LIN {X 0,Y 581.296,Z 726.906,A -85,B 0,C 180,E1 9487.47,E2 9487.47} C_VEL
LIN {X 0,Y 571.469,Z 707.643,A -85,B 0,C 180,E1 9488.58,E2 9488.58} C_VEL
LIN {X 0,Y 571.367,Z 707.31,A -85,B 0,C 180,E1 9494.263,E2 9494.263} C_VEL
LIN {X 0,Y 571.407,Z 707.31,A -85,B 0,C 180,E1 9500.466,E2 9500.466} C_VEL
LIN {X 0,Y 571.477,Z 707.31,A -85,B 0,C 180,E1 9506.158,E2 9506.158} C_VEL
LIN {X 0,Y 571.546,Z 707.31,A -85,B 0,C 180,E1 9511.491,E2 9511.491} C_VEL
LIN {X 0,Y 571.588,Z 707.31,A -85,B 0,C 180,E1 9516.564,E2 9516.564} C_VEL
LIN {X 0,Y 571.677,Z 707.31,A -85,B 0,C 180,E1 9522.611,E2 9522.611} C_VEL
LIN {X 0,Y 572.124,Z 707.31,A -85,B 0,C 180,E1 9528.533,E2 9528.533} C_VEL
LIN {X 0,Y 572.269,Z 707.31,A -85,B 0,C 180,E1 9533.917,E2 9533.917} C_VEL
LIN {X 0,Y 572.201,Z 707.31,A -85,B 0,C 180,E1 9539.997,E2 9539.997} C_VEL
LIN {X 0,Y 572.109,Z 707.31,A -85,B 0,C 180,E1 9546.079,E2 9546.079} C_VEL
LIN {X 0,Y 572.048,Z 707.31,A -85,B 0,C 180,E1 9551.43,E2 9551.43} C_VEL
LIN {X 0,Y 571.675,Z 707.31,A -85,B 0,C 180,E1 9557.388,E2 9557.388} C_VEL
LIN {X 0,Y 571.56,Z 707.31,A -85,B 0,C 180,E1 9563.431,E2 9563.431} C_VEL
LIN {X 0,Y 571.547,Z 707.31,A -85,B 0,C 180,E1 9568.958,E2 9568.958} C_VEL
LIN {X 0,Y 571.47,Z 707.31,A -85,B 0,C 180,E1 9574.709,E2 9574.709} C_VEL
LIN {X 0,Y 571.379,Z 707.31,A -85,B 0,C 180,E1 9579.723,E2 9579.723} C_VEL
LIN {X 0,Y 571.332,Z 707.31,A -85,B 0,C 180,E1 9585.733,E2 9585.733} C_VEL
LIN {X 0,Y 571.387,Z 707.31,A -85,B 0,C 180,E1 9588.976,E2 9588.976} C_VEL
LIN {X 0,Y 578.42,Z 721.819,A -85,B 0,C 180,E1 9589.801,E2 9589.801} C_VEL
LIN {X 0,Y 603.039,Z 770.669,A -85,B 0,C 180,E1 9592.453,E2 9592.453} C_VEL
LIN {X 0,Y 600.05,Z 820.289,A -85,B 0,C 180,E1 9593.653,E2 9593.653} C_VEL
LIN {X 0,Y 598.7,Z 837.933,A -85,B 0,C 180,E1 9594.27,E2 9594.27} C_VEL
LIN {X 0,Y 593.828,Z 854.218,A -85,B 0,C 180,E1 9594.704,E2 9594.704} C_VEL
LIN {X 0,Y 588.685,Z 870.067,A -85,B 0,C 180,E1 9595.207,E2 9595.207} C_VEL
LIN {X 0,Y 583.535,Z 912.903,A -85,B 0,C 180,E1 9597.679,E2 9597.679} C_VEL
LIN {X 0,Y 578.202,Z 952.807,A -85,B 0,C 180,E1 9600.781,E2 9600.781} C_VEL
LIN {X 0,Y 573.288,Z 989.217,A -85,B 0,C 180,E1 9604.529,E2 9604.529} C_VEL
LIN {X 0,Y 569.458,Z 1019.706,A -85,B 0,C 180,E1 9608.644,E2 9608.644} C_VEL
LIN {X 0,Y 566.797,Z 1045.546,A -85,B 0,C 180,E1 9613.296,E2 9613.296} C_VEL
LIN {X 0,Y 565.422,Z 1063.972,A -85,B 0,C 180,E1 9617.923,E2 9617.923} C_VEL
LIN {X 0,Y 564.867,Z 1075.583,A -85,B 0,C 180,E1 9622.291,E2 9622.291} C_VEL
LIN {X 0,Y 564.721,Z 1080.643,A -85,B 0,C 180,E1 9625.382,E2 9625.382} C_VEL
LIN {X 0,Y 564.787,Z 1083.5,A -85,B 0,C 180,E1 9629.999,E2 9629.999} C_VEL
LIN {X 0,Y 564.751,Z 1080.646,A -85,B 0,C 180,E1 9634.617,E2 9634.617} C_VEL
LIN {X 0,Y 564.884,Z 1073.99,A -85,B 0,C 180,E1 9638.484,E2 9638.484} C_VEL
LIN {X 0,Y 565.598,Z 1060.203,A -85,B 0,C 180,E1 9643.163,E2 9643.163} C_VEL
LIN {X 0,Y 567.063,Z 1041.597,A -85,B 0,C 180,E1 9647.495,E2 9647.495} C_VEL
LIN {X 0,Y 569.661,Z 1017.405,A -85,B 0,C 180,E1 9651.696,E2 9651.696} C_VEL
LIN {X 0,Y 573.518,Z 986.806,A -85,B 0,C 180,E1 9655.747,E2 9655.747} C_VEL
LIN {X 0,Y 578.55,Z 950.559,A -85,B 0,C 180,E1 9659.413,E2 9659.413} C_VEL
LIN {X 0,Y 584.004,Z 910.777,A -85,B 0,C 180,E1 9662.474,E2 9662.474} C_VEL
LIN {X 0,Y 589.211,Z 868.238,A -85,B 0,C 180,E1 9664.906,E2 9664.906} C_VEL
LIN {X 0,Y 593.615,Z 824.295,A -85,B 0,C 180,E1 9666.688,E2 9666.688} C_VEL
LIN {X 0,Y 596.654,Z 780.659,A -85,B 0,C 180,E1 9667.85,E2 9667.85} C_VEL
LIN {X 0,Y 596.255,Z 771.433,A -85,B 0,C 180,E1 9668.098,E2 9668.098} C_VEL
LIN {X 0,Y 574.83,Z 728.644,A -85,B 0,C 180,E1 9670.579,E2 9670.579} C_VEL
LIN {X 0,Y 563.718,Z 709.225,A -85,B 0,C 180,E1 9671.902,E2 9671.902} C_VEL
LIN {X 0,Y 563.489,Z 707.31,A -85,B 0,C 180,E1 9672.019,E2 9672.019} C_VEL
LIN {X 0,Y 563.451,Z 707.31,A -85,B 0,C 180,E1 9677.754,E2 9677.754} C_VEL
LIN {X 0,Y 563.526,Z 707.31,A -85,B 0,C 180,E1 9683.778,E2 9683.778} C_VEL
LIN {X 0,Y 563.666,Z 707.31,A -85,B 0,C 180,E1 9689.35,E2 9689.35} C_VEL
LIN {X 0,Y 563.629,Z 707.31,A -85,B 0,C 180,E1 9694.524,E2 9694.524} C_VEL
LIN {X 0,Y 563.692,Z 707.31,A -85,B 0,C 180,E1 9700.205,E2 9700.205} C_VEL
LIN {X 0,Y 563.965,Z 707.31,A -85,B 0,C 180,E1 9706.008,E2 9706.008} C_VEL
LIN {X 0,Y 564.245,Z 707.31,A -85,B 0,C 180,E1 9710.73,E2 9710.73} C_VEL
LIN {X 0,Y 563.991,Z 707.31,A -85,B 0,C 180,E1 9715.379,E2 9715.379} C_VEL
LIN {X 0,Y 564.275,Z 707.31,A -85,B 0,C 180,E1 9720.003,E2 9720.003} C_VEL
LIN {X 0,Y 564.043,Z 707.31,A -85,B 0,C 180,E1 9726.25,E2 9726.25} C_VEL
LIN {X 0,Y 564.054,Z 707.31,A -85,B 0,C 180,E1 9732.414,E2 9732.414} C_VEL
LIN {X 0,Y 563.768,Z 707.31,A -85,B 0,C 180,E1 9738.82,E2 9738.82} C_VEL
LIN {X 0,Y 563.719,Z 707.31,A -85,B 0,C 180,E1 9743.939,E2 9743.939} C_VEL
LIN {X 0,Y 563.492,Z 707.31,A -85,B 0,C 180,E1 9748.955,E2 9748.955} C_VEL
LIN {X 0,Y 563.465,Z 707.31,A -85,B 0,C 180,E1 9754.39,E2 9754.39} C_VEL
LIN {X 0,Y 563.457,Z 707.31,A -85,B 0,C 180,E1 9760.204,E2 9760.204} C_VEL
LIN {X 0,Y 563.487,Z 707.4,A -85,B 0,C 180,E1 9766.379,E2 9766.379} C_VEL
LIN {X 0,Y 568.232,Z 717.353,A -85,B 0,C 180,E1 9766.983,E2 9766.983} C_VEL
LIN {X 0,Y 588.613,Z 755.907,A -85,B 0,C 180,E1 9769.479,E2 9769.479} C_VEL
LIN {X 0,Y 595.824,Z 774.73,A -85,B 0,C 180,E1 9770.57,E2 9770.57} C_VEL
LIN {X 0,Y 591.999,Z 820.472,A -85,B 0,C 180,E1 9772.096,E2 9772.096} C_VEL
LIN {X 0,Y 587.146,Z 862.961,A -85,B 0,C 180,E1 9774.17,E2 9774.17} C_VEL
LIN {X 0,Y 582.133,Z 901.788,A -85,B 0,C 180,E1 9776.757,E2 9776.757} C_VEL
LIN {X 0,Y 576.775,Z 939.323,A -85,B 0,C 180,E1 9780.054,E2 9780.054} C_VEL
LIN {X 0,Y 572.225,Z 972.486,A -85,B 0,C 180,E1 9783.881,E2 9783.881} C_VEL
LIN {X 0,Y 568.66,Z 1000.305,A -85,B 0,C 180,E1 9788.095,E2 9788.095} C_VEL
LIN {X 0,Y 566.274,Z 1023.607,A -85,B 0,C 180,E1 9792.881,E2 9792.881} C_VEL
LIN {X 0,Y 565.16,Z 1039.587,A -85,B 0,C 180,E1 9797.614,E2 9797.614} C_VEL
LIN {X 0,Y 564.745,Z 1049.246,A -85,B 0,C 180,E1 9802.29,E2 9802.29} C_VEL
LIN {X 0,Y 564.561,Z 1053.277,A -85,B 0,C 180,E1 9806.923,E2 9806.923} C_VEL
LIN {X 0,Y 564.853,Z 1052.901,A -85,B 0,C 180,E1 9810.001,E2 9810.001} C_VEL
LIN {X 0,Y 564.793,Z 1047.709,A -85,B 0,C 180,E1 9814.618,E2 9814.618} C_VEL
LIN {X 0,Y 565.152,Z 1037.925,A -85,B 0,C 180,E1 9818.87,E2 9818.87} C_VEL
LIN {X 0,Y 566.241,Z 1023.115,A -85,B 0,C 180,E1 9823.149,E2 9823.149} C_VEL
LIN {X 0,Y 568.566,Z 1000.113,A -85,B 0,C 180,E1 9827.85,E2 9827.85} C_VEL
LIN {X 0,Y 572.256,Z 971.194,A -85,B 0,C 180,E1 9832.202,E2 9832.202} C_VEL
LIN {X 0,Y 577.134,Z 936.917,A -85,B 0,C 180,E1 9836.093,E2 9836.093} C_VEL
LIN {X 0,Y 582.635,Z 897.836,A -85,B 0,C 180,E1 9839.435,E2 9839.435} C_VEL
LIN {X 0,Y 588.021,Z 856.086,A -85,B 0,C 180,E1 9842.09,E2 9842.09} C_VEL
LIN {X 0,Y 592.591,Z 812.427,A -85,B 0,C 180,E1 9844.087,E2 9844.087} C_VEL
LIN {X 0,Y 594.966,Z 772.076,A -85,B 0,C 180,E1 9845.404,E2 9845.404} C_VEL
LIN {X 0,Y 574.604,Z 728.871,A -85,B 0,C 180,E1 9847.981,E2 9847.981} C_VEL
LIN {X 0,Y 563.598,Z 708.617,A -85,B 0,C 180,E1 9849.24,E2 9849.24} C_VEL
LIN {X 0,Y 563.51,Z 707.31,A -85,B 0,C 180,E1 9849.325,E2 9849.325} C_VEL
LIN {X 0,Y 563.489,Z 707.31,A -85,B 0,C 180,E1 9855.632,E2 9855.632} C_VEL
LIN {X 0,Y 563.458,Z 707.31,A -85,B 0,C 180,E1 9861.785,E2 9861.785} C_VEL
LIN {X 0,Y 563.6,Z 707.31,A -85,B 0,C 180,E1 9867.466,E2 9867.466} C_VEL
LIN {X 0,Y 563.638,Z 707.31,A -85,B 0,C 180,E1 9872.8,E2 9872.8} C_VEL
LIN {X 0,Y 563.701,Z 707.31,A -85,B 0,C 180,E1 9877.889,E2 9877.889} C_VEL
LIN {X 0,Y 563.962,Z 707.31,A -85,B 0,C 180,E1 9884.41,E2 9884.41} C_VEL
LIN {X 0,Y 564.262,Z 707.31,A -85,B 0,C 180,E1 9889.162,E2 9889.162} C_VEL
LIN {X 0,Y 564.354,Z 707.31,A -85,B 0,C 180,E1 9895.377,E2 9895.377} C_VEL
LIN {X 0,Y 564.428,Z 707.31,A -85,B 0,C 180,E1 9901.536,E2 9901.536} C_VEL
LIN {X 0,Y 564.373,Z 707.31,A -85,B 0,C 180,E1 9907.713,E2 9907.713} C_VEL
LIN {X 0,Y 564.094,Z 707.31,A -85,B 0,C 180,E1 9912.407,E2 9912.407} C_VEL
LIN {X 0,Y 563.812,Z 707.31,A -85,B 0,C 180,E1 9917.194,E2 9917.194} C_VEL
LIN {X 0,Y 563.661,Z 707.31,A -85,B 0,C 180,E1 9922.107,E2 9922.107} C_VEL
LIN {X 0,Y 563.635,Z 707.31,A -85,B 0,C 180,E1 9927.47,E2 9927.47} C_VEL
LIN {X 0,Y 563.558,Z 707.31,A -85,B 0,C 180,E1 9933.53,E2 9933.53} C_VEL
LIN {X 0,Y 563.439,Z 707.31,A -85,B 0,C 180,E1 9938.741,E2 9938.741} C_VEL
LIN {X 0,Y 563.438,Z 707.31,A -85,B 0,C 180,E1 9944.365,E2 9944.365} C_VEL
LIN {X 0,Y 563.428,Z 707.31,A -85,B 0,C 180,E1 9948.305,E2 9948.305} C_VEL
LIN {X 0,Y 567.631,Z 716.59,A -85,B 0,C 180,E1 9948.821,E2 9948.821} C_VEL
LIN {X 0,Y 593.946,Z 767.38,A -85,B 0,C 180,E1 9951.737,E2 9951.737} C_VEL
LIN {X 0,Y 596.749,Z 775.021,A -85,B 0,C 180,E1 9952.103,E2 9952.103} C_VEL
LIN {X 0,Y 593.487,Z 821.368,A -85,B 0,C 180,E1 9953.247,E2 9953.247} C_VEL
LIN {X 0,Y 588.967,Z 867.48,A -85,B 0,C 180,E1 9955.075,E2 9955.075} C_VEL
LIN {X 0,Y 588.685,Z 870.067,A -85,B 0,C 180,E1 9955.207,E2 9955.207} C_VEL
LIN {X 0,Y 583.54,Z 885.733,A -85,B 0,C 180,E1 9955.813,E2 9955.813} C_VEL
LIN {X 0,Y 578.291,Z 900.889,A -85,B 0,C 180,E1 9956.497,E2 9956.497} C_VEL
LIN {X 0,Y 572.773,Z 940.932,A -85,B 0,C 180,E1 9959.383,E2 9959.383} C_VEL
LIN {X 0,Y 567.644,Z 976.893,A -85,B 0,C 180,E1 9962.794,E2 9962.794} C_VEL
LIN {X 0,Y 562.952,Z 1010.727,A -85,B 0,C 180,E1 9967.025,E2 9967.025} C_VEL
LIN {X 0,Y 559.825,Z 1036.76,A -85,B 0,C 180,E1 9971.327,E2 9971.327} C_VEL
LIN {X 0,Y 558.022,Z 1057.049,A -85,B 0,C 180,E1 9975.852,E2 9975.852} C_VEL
LIN {X 0,Y 557.265,Z 1069.881,A -85,B 0,C 180,E1 9979.818,E2 9979.818} C_VEL
LIN {X 0,Y 556.926,Z 1079.473,A -85,B 0,C 180,E1 9984.534,E2 9984.534} C_VEL
LIN {X 0,Y 556.74,Z 1083.028,A -85,B 0,C 180,E1 9988.44,E2 9988.44} C_VEL
LIN {X 0,Y 556.9,Z 1082.064,A -85,B 0,C 180,E1 9993.119,E2 9993.119} C_VEL
LIN {X 0,Y 556.912,Z 1076.928,A -85,B 0,C 180,E1 9997.05,E2 9997.05} C_VEL
LIN {X 0,Y 557.572,Z 1064.769,A -85,B 0,C 180,E1 10001.94,E2 10001.94} C_VEL
LIN {X 0,Y 558.858,Z 1047.085,A -85,B 0,C 180,E1 10006.541,E2 10006.541} C_VEL
LIN {X 0,Y 561.141,Z 1024.724,A -85,B 0,C 180,E1 10010.796,E2 10010.796} C_VEL
LIN {X 0,Y 564.747,Z 997.074,A -85,B 0,C 180,E1 10014.819,E2 10014.819} C_VEL
LIN {X 0,Y 569.574,Z 963.246,A -85,B 0,C 180,E1 10018.613,E2 10018.613} C_VEL
LIN {X 0,Y 575.241,Z 924.394,A -85,B 0,C 180,E1 10021.937,E2 10021.937} C_VEL
LIN {X 0,Y 580.9,Z 882.32,A -85,B 0,C 180,E1 10024.631,E2 10024.631} C_VEL
LIN {X 0,Y 585.988,Z 836.937,A -85,B 0,C 180,E1 10026.715,E2 10026.715} C_VEL
LIN {X 0,Y 590.009,Z 788.172,A -85,B 0,C 180,E1 10028.171,E2 10028.171} C_VEL
LIN {X 0,Y 590.101,Z 774.484,A -85,B 0,C 180,E1 10028.501,E2 10028.501} C_VEL
LIN {X 0,Y 569.808,Z 733.63,A -85,B 0,C 180,E1 10030.939,E2 10030.939} C_VEL
LIN {X 0,Y 555.597,Z 707.982,A -85,B 0,C 180,E1 10032.696,E2 10032.696} C_VEL
LIN {X 0,Y 555.528,Z 707.31,A -85,B 0,C 180,E1 10037.435,E2 10037.435} C_VEL
LIN {X 0,Y 555.525,Z 707.31,A -85,B 0,C 180,E1 10043.125,E2 10043.125} C_VEL
LIN {X 0,Y 555.685,Z 707.31,A -85,B 0,C 180,E1 10048.796,E2 10048.796} C_VEL
LIN {X 0,Y 555.7,Z 707.31,A -85,B 0,C 180,E1 10054.145,E2 10054.145} C_VEL
LIN {X 0,Y 555.737,Z 707.31,A -85,B 0,C 180,E1 10059.241,E2 10059.241} C_VEL
LIN {X 0,Y 555.944,Z 707.31,A -85,B 0,C 180,E1 10064.185,E2 10064.185} C_VEL
LIN {X 0,Y 556.277,Z 707.31,A -85,B 0,C 180,E1 10069.01,E2 10069.01} C_VEL
LIN {X 0,Y 556.324,Z 707.31,A -85,B 0,C 180,E1 10073.748,E2 10073.748} C_VEL
LIN {X 0,Y 556.377,Z 707.31,A -85,B 0,C 180,E1 10080.003,E2 10080.003} C_VEL
LIN {X 0,Y 556.165,Z 707.31,A -85,B 0,C 180,E1 10086.26,E2 10086.26} C_VEL
LIN {X 0,Y 556.135,Z 707.31,A -85,B 0,C 180,E1 10092.594,E2 10092.594} C_VEL
LIN {X 0,Y 555.863,Z 707.31,A -85,B 0,C 180,E1 10099.098,E2 10099.098} C_VEL
LIN {X 0,Y 555.795,Z 707.31,A -85,B 0,C 180,E1 10104.144,E2 10104.144} C_VEL
LIN {X 0,Y 555.57,Z 707.31,A -85,B 0,C 180,E1 10109.408,E2 10109.408} C_VEL
LIN {X 0,Y 555.51,Z 707.31,A -85,B 0,C 180,E1 10115.078,E2 10115.078} C_VEL
LIN {X 0,Y 555.577,Z 707.31,A -85,B 0,C 180,E1 10120.895,E2 10120.895} C_VEL
LIN {X 0,Y 555.577,Z 707.31,A -85,B 0,C 180,E1 10125.616,E2 10125.616} C_VEL
LIN {X 0,Y 558.06,Z 713.056,A -85,B 0,C 180,E1 10125.963,E2 10125.963} C_VEL
LIN {X 0,Y 581.404,Z 756.646,A -85,B 0,C 180,E1 10128.91,E2 10128.91} C_VEL
LIN {X 0,Y 589.506,Z 776.851,A -85,B 0,C 180,E1 10130.144,E2 10130.144} C_VEL
LIN {X 0,Y 585.345,Z 823.942,A -85,B 0,C 180,E1 10131.769,E2 10131.769} C_VEL
LIN {X 0,Y 579.997,Z 867.511,A -85,B 0,C 180,E1 10133.977,E2 10133.977} C_VEL
LIN {X 0,Y 574.534,Z 907.094,A -85,B 0,C 180,E1 10136.74,E2 10136.74} C_VEL
LIN {X 0,Y 569.332,Z 941.576,A -85,B 0,C 180,E1 10139.884,E2 10139.884} C_VEL
LIN {X 0,Y 564.636,Z 973.931,A -85,B 0,C 180,E1 10143.715,E2 10143.715} C_VEL
LIN {X 0,Y 560.916,Z 1001.672,A -85,B 0,C 180,E1 10148.025,E2 10148.025} C_VEL
LIN {X 0,Y 558.559,Z 1023.705,A -85,B 0,C 180,E1 10152.637,E2 10152.637} C_VEL
LIN {X 0,Y 557.31,Z 1039.716,A -85,B 0,C 180,E1 10157.437,E2 10157.437} C_VEL
LIN {X 0,Y 556.848,Z 1049.414,A -85,B 0,C 180,E1 10162.18,E2 10162.18} C_VEL
LIN {X 0,Y 556.662,Z 1053.427,A -85,B 0,C 180,E1 10166.88,E2 10166.88} C_VEL
LIN {X 0,Y 556.953,Z 1053.075,A -85,B 0,C 180,E1 10170.001,E2 10170.001} C_VEL
LIN {X 0,Y 556.919,Z 1047.964,A -85,B 0,C 180,E1 10174.683,E2 10174.683} C_VEL
LIN {X 0,Y 557.311,Z 1038.221,A -85,B 0,C 180,E1 10178.996,E2 10178.996} C_VEL
LIN {X 0,Y 558.48,Z 1023.454,A -85,B 0,C 180,E1 10183.336,E2 10183.336} C_VEL
LIN {X 0,Y 560.934,Z 1000.505,A -85,B 0,C 180,E1 10188.101,E2 10188.101} C_VEL
LIN {X 0,Y 564.914,Z 971.057,A -85,B 0,C 180,E1 10192.585,E2 10192.585} C_VEL
LIN {X 0,Y 569.98,Z 937.4,A -85,B 0,C 180,E1 10196.445,E2 10196.445} C_VEL
LIN {X 0,Y 575.737,Z 898.468,A -85,B 0,C 180,E1 10199.814,E2 10199.814} C_VEL
LIN {X 0,Y 581.382,Z 856.241,A -85,B 0,C 180,E1 10202.529,E2 10202.529} C_VEL
LIN {X 0,Y 586.141,Z 812.729,A -85,B 0,C 180,E1 10204.533,E2 10204.533} C_VEL
LIN {X 0,Y 588.638,Z 775.079,A -85,B 0,C 180,E1 10205.784,E2 10205.784} C_VEL
LIN {X 0,Y 568.389,Z 731.925,A -85,B 0,C 180,E1 10208.442,E2 10208.442} C_VEL
LIN {X 0,Y 555.589,Z 707.992,A -85,B 0,C 180,E1 10209.964,E2 10209.964} C_VEL
LIN {X 0,Y 555.567,Z 707.31,A -85,B 0,C 180,E1 10215.17,E2 10215.17} C_VEL
LIN {X 0,Y 555.573,Z 707.31,A -85,B 0,C 180,E1 10221.142,E2 10221.142} C_VEL
LIN {X 0,Y 555.69,Z 707.31,A -85,B 0,C 180,E1 10227.715,E2 10227.715} C_VEL
LIN {X 0,Y 555.716,Z 707.31,A -85,B 0,C 180,E1 10232.379,E2 10232.379} C_VEL
LIN {X 0,Y 555.805,Z 707.31,A -85,B 0,C 180,E1 10237.975,E2 10237.975} C_VEL
LIN {X 0,Y 556.014,Z 707.31,A -85,B 0,C 180,E1 10244.181,E2 10244.181} C_VEL
LIN {X 0,Y 556.338,Z 707.31,A -85,B 0,C 180,E1 10249.005,E2 10249.005} C_VEL
LIN {X 0,Y 556.454,Z 707.31,A -85,B 0,C 180,E1 10255.311,E2 10255.311} C_VEL
LIN {X 0,Y 556.525,Z 707.31,A -85,B 0,C 180,E1 10261.557,E2 10261.557} C_VEL
LIN {X 0,Y 556.45,Z 707.31,A -85,B 0,C 180,E1 10267.823,E2 10267.823} C_VEL
LIN {X 0,Y 556.173,Z 707.31,A -85,B 0,C 180,E1 10272.587,E2 10272.587} C_VEL
LIN {X 0,Y 555.877,Z 707.31,A -85,B 0,C 180,E1 10277.447,E2 10277.447} C_VEL
LIN {X 0,Y 555.728,Z 707.31,A -85,B 0,C 180,E1 10282.44,E2 10282.44} C_VEL
LIN {X 0,Y 555.731,Z 707.31,A -85,B 0,C 180,E1 10287.614,E2 10287.614} C_VEL
LIN {X 0,Y 555.674,Z 707.31,A -85,B 0,C 180,E1 10293.05,E2 10293.05} C_VEL
LIN {X 0,Y 555.552,Z 707.31,A -85,B 0,C 180,E1 10298.853,E2 10298.853} C_VEL
LIN {X 0,Y 555.521,Z 707.31,A -85,B 0,C 180,E1 10305.169,E2 10305.169} C_VEL
LIN {X 0,Y 555.576,Z 707.871,A -85,B 0,C 180,E1 10307.615,E2 10307.615} C_VEL
LIN {X 0,Y 587.663,Z 770.146,A -85,B 0,C 180,E1 10311.319,E2 10311.319} C_VEL
LIN {X 0,Y 590.284,Z 778.186,A -85,B 0,C 180,E1 10311.704,E2 10311.704} C_VEL
LIN {X 0,Y 586.967,Z 822.15,A -85,B 0,C 180,E1 10312.822,E2 10312.822} C_VEL
LIN {X 0,Y 582.334,Z 867.091,A -85,B 0,C 180,E1 10314.618,E2 10314.618} C_VEL
LIN {X 0,Y 578.291,Z 900.889,A -85,B 0,C 180,E1 10316.497,E2 10316.497} C_VEL
LIN {X 0,Y 572.812,Z 915.73,A -85,B 0,C 180,E1 10317.264,E2 10317.264} C_VEL
LIN {X 0,Y 567.334,Z 930.006,A -85,B 0,C 180,E1 10318.111,E2 10318.111} C_VEL
LIN {X 0,Y 561.9,Z 966.272,A -85,B 0,C 180,E1 10321.325,E2 10321.325} C_VEL
LIN {X 0,Y 556.905,Z 1000.251,A -85,B 0,C 180,E1 10325.267,E2 10325.267} C_VEL
LIN {X 0,Y 552.897,Z 1029.524,A -85,B 0,C 180,E1 10329.755,E2 10329.755} C_VEL
LIN {X 0,Y 550.596,Z 1052.088,A -85,B 0,C 180,E1 10334.416,E2 10334.416} C_VEL
LIN {X 0,Y 549.455,Z 1068.58,A -85,B 0,C 180,E1 10339.27,E2 10339.27} C_VEL
LIN {X 0,Y 549.014,Z 1078.03,A -85,B 0,C 180,E1 10343.66,E2 10343.66} C_VEL
LIN {X 0,Y 548.841,Z 1082.818,A -85,B 0,C 180,E1 10348.417,E2 10348.417} C_VEL
LIN {X 0,Y 548.994,Z 1081.852,A -85,B 0,C 180,E1 10353.164,E2 10353.164} C_VEL
LIN {X 0,Y 549.042,Z 1076.905,A -85,B 0,C 180,E1 10357.054,E2 10357.054} C_VEL
LIN {X 0,Y 549.699,Z 1064.552,A -85,B 0,C 180,E1 10362.113,E2 10362.113} C_VEL
LIN {X 0,Y 551.063,Z 1046.865,A -85,B 0,C 180,E1 10366.782,E2 10366.782} C_VEL
LIN {X 0,Y 553.341,Z 1025.941,A -85,B 0,C 180,E1 10370.855,E2 10370.855} C_VEL
LIN {X 0,Y 557.322,Z 997.111,A -85,B 0,C 180,E1 10375.141,E2 10375.141} C_VEL
LIN {X 0,Y 562.46,Z 963.098,A -85,B 0,C 180,E1 10379.009,E2 10379.009} C_VEL
LIN {X 0,Y 568.337,Z 924.623,A -85,B 0,C 180,E1 10382.346,E2 10382.346} C_VEL
LIN {X 0,Y 574.484,Z 881.133,A -85,B 0,C 180,E1 10385.147,E2 10385.147} C_VEL
LIN {X 0,Y 579.793,Z 835.679,A -85,B 0,C 180,E1 10387.235,E2 10387.235} C_VEL
LIN {X 0,Y 583.979,Z 786.474,A -85,B 0,C 180,E1 10388.694,E2 10388.694} C_VEL
LIN {X 0,Y 583.669,Z 776.789,A -85,B 0,C 180,E1 10388.957,E2 10388.957} C_VEL
LIN {X 0,Y 563.575,Z 736.476,A -85,B 0,C 180,E1 10391.455,E2 10391.455} C_VEL
LIN {X 0,Y 547.702,Z 708.531,A -85,B 0,C 180,E1 10393.471,E2 10393.471} C_VEL
LIN {X 0,Y 547.578,Z 707.31,A -85,B 0,C 180,E1 10393.618,E2 10393.618} C_VEL
LIN {X 0,Y 547.583,Z 707.31,A -85,B 0,C 180,E1 10398.385,E2 10398.385} C_VEL
LIN {X 0,Y 547.62,Z 707.31,A -85,B 0,C 180,E1 10404.475,E2 10404.475} C_VEL
LIN {X 0,Y 547.768,Z 707.31,A -85,B 0,C 180,E1 10410.138,E2 10410.138} C_VEL
LIN {X 0,Y 547.793,Z 707.31,A -85,B 0,C 180,E1 10415.908,E2 10415.908} C_VEL
LIN {X 0,Y 547.925,Z 707.31,A -85,B 0,C 180,E1 10422.292,E2 10422.292} C_VEL
LIN {X 0,Y 548.224,Z 707.31,A -85,B 0,C 180,E1 10427.227,E2 10427.227} C_VEL
LIN {X 0,Y 548.536,Z 707.31,A -85,B 0,C 180,E1 10432.063,E2 10432.063} C_VEL
LIN {X 0,Y 548.611,Z 707.31,A -85,B 0,C 180,E1 10438.42,E2 10438.42} C_VEL
LIN {X 0,Y 548.349,Z 707.31,A -85,B 0,C 180,E1 10444.758,E2 10444.758} C_VEL
LIN {X 0,Y 548.265,Z 707.31,A -85,B 0,C 180,E1 10451.159,E2 10451.159} C_VEL
LIN {X 0,Y 547.967,Z 707.31,A -85,B 0,C 180,E1 10456.057,E2 10456.057} C_VEL
LIN {X 0,Y 547.968,Z 707.31,A -85,B 0,C 180,E1 10461.073,E2 10461.073} C_VEL
LIN {X 0,Y 547.717,Z 707.31,A -85,B 0,C 180,E1 10466.278,E2 10466.278} C_VEL
LIN {X 0,Y 547.629,Z 707.31,A -85,B 0,C 180,E1 10471.723,E2 10471.723} C_VEL
LIN {X 0,Y 547.603,Z 707.31,A -85,B 0,C 180,E1 10477.507,E2 10477.507} C_VEL
LIN {X 0,Y 547.603,Z 707.31,A -85,B 0,C 180,E1 10483.779,E2 10483.779} C_VEL
LIN {X 0,Y 547.68,Z 707.324,A -85,B 0,C 180,E1 10484.839,E2 10484.839} C_VEL
LIN {X 0,Y 550.095,Z 713.01,A -85,B 0,C 180,E1 10485.183,E2 10485.183} C_VEL
LIN {X 0,Y 573.971,Z 756.758,A -85,B 0,C 180,E1 10488.285,E2 10488.285} C_VEL
LIN {X 0,Y 583.063,Z 780.371,A -85,B 0,C 180,E1 10489.751,E2 10489.751} C_VEL
LIN {X 0,Y 578.776,Z 826.32,A -85,B 0,C 180,E1 10491.386,E2 10491.386} C_VEL
LIN {X 0,Y 572.937,Z 871.717,A -85,B 0,C 180,E1 10493.763,E2 10493.763} C_VEL
LIN {X 0,Y 566.905,Z 912.975,A -85,B 0,C 180,E1 10496.772,E2 10496.772} C_VEL
LIN {X 0,Y 560.867,Z 950.348,A -85,B 0,C 180,E1 10500.406,E2 10500.406} C_VEL
LIN {X 0,Y 555.874,Z 982.675,A -85,B 0,C 180,E1 10504.573,E2 10504.573} C_VEL
LIN {X 0,Y 552.324,Z 1009.098,A -85,B 0,C 180,E1 10509.104,E2 10509.104} C_VEL
LIN {X 0,Y 550.173,Z 1029.909,A -85,B 0,C 180,E1 10514.013,E2 10514.013} C_VEL
LIN {X 0,Y 549.236,Z 1043.752,A -85,B 0,C 180,E1 10518.865,E2 10518.865} C_VEL
LIN {X 0,Y 548.88,Z 1051.543,A -85,B 0,C 180,E1 10523.66,E2 10523.66} C_VEL
LIN {X 0,Y 548.805,Z 1053.77,A -85,B 0,C 180,E1 10528.418,E2 10528.418} C_VEL
LIN {X 0,Y 548.889,Z 1052.252,A -85,B 0,C 180,E1 10531.583,E2 10531.583} C_VEL
LIN {X 0,Y 549.148,Z 1045.254,A -85,B 0,C 180,E1 10536.338,E2 10536.338} C_VEL
LIN {X 0,Y 549.976,Z 1032.45,A -85,B 0,C 180,E1 10541.121,E2 10541.121} C_VEL
LIN {X 0,Y 551.697,Z 1015.103,A -85,B 0,C 180,E1 10545.535,E2 10545.535} C_VEL
LIN {X 0,Y 554.703,Z 991.422,A -85,B 0,C 180,E1 10549.968,E2 10549.968} C_VEL
LIN {X 0,Y 559.225,Z 960.957,A -85,B 0,C 180,E1 10554.242,E2 10554.242} C_VEL
LIN {X 0,Y 564.882,Z 924.639,A -85,B 0,C 180,E1 10558.077,E2 10558.077} C_VEL
LIN {X 0,Y 570.815,Z 885.579,A -85,B 0,C 180,E1 10561.178,E2 10561.178} C_VEL
LIN {X 0,Y 576.541,Z 841.067,A -85,B 0,C 180,E1 10563.781,E2 10563.781} C_VEL
LIN {X 0,Y 581.46,Z 793.951,A -85,B 0,C 180,E1 10565.671,E2 10565.671} C_VEL
LIN {X 0,Y 582.161,Z 777.652,A -85,B 0,C 180,E1 10566.198,E2 10566.198} C_VEL
LIN {X 0,Y 561.584,Z 733.626,A -85,B 0,C 180,E1 10568.992,E2 10568.992} C_VEL
LIN {X 0,Y 547.671,Z 708.055,A -85,B 0,C 180,E1 10570.697,E2 10570.697} C_VEL
LIN {X 0,Y 547.608,Z 707.31,A -85,B 0,C 180,E1 10576.222,E2 10576.222} C_VEL
LIN {X 0,Y 547.629,Z 707.31,A -85,B 0,C 180,E1 10582.495,E2 10582.495} C_VEL
LIN {X 0,Y 547.775,Z 707.31,A -85,B 0,C 180,E1 10589.05,E2 10589.05} C_VEL
LIN {X 0,Y 547.77,Z 707.31,A -85,B 0,C 180,E1 10593.725,E2 10593.725} C_VEL
LIN {X 0,Y 547.854,Z 707.31,A -85,B 0,C 180,E1 10600.131,E2 10600.131} C_VEL
LIN {X 0,Y 548.23,Z 707.31,A -85,B 0,C 180,E1 10605.592,E2 10605.592} C_VEL
LIN {X 0,Y 548.44,Z 707.31,A -85,B 0,C 180,E1 10610.454,E2 10610.454} C_VEL
LIN {X 0,Y 548.546,Z 707.31,A -85,B 0,C 180,E1 10615.243,E2 10615.243} C_VEL
LIN {X 0,Y 548.613,Z 707.31,A -85,B 0,C 180,E1 10621.58,E2 10621.58} C_VEL
LIN {X 0,Y 548.55,Z 707.31,A -85,B 0,C 180,E1 10627.937,E2 10627.937} C_VEL
LIN {X 0,Y 548.237,Z 707.31,A -85,B 0,C 180,E1 10632.772,E2 10632.772} C_VEL
LIN {X 0,Y 547.933,Z 707.31,A -85,B 0,C 180,E1 10637.708,E2 10637.708} C_VEL
LIN {X 0,Y 547.804,Z 707.31,A -85,B 0,C 180,E1 10644.091,E2 10644.091} C_VEL
LIN {X 0,Y 547.761,Z 707.31,A -85,B 0,C 180,E1 10649.862,E2 10649.862} C_VEL
LIN {X 0,Y 547.627,Z 707.31,A -85,B 0,C 180,E1 10655.525,E2 10655.525} C_VEL
LIN {X 0,Y 547.593,Z 707.31,A -85,B 0,C 180,E1 10661.651,E2 10661.651} C_VEL
LIN {X 0,Y 547.6,Z 707.31,A -85,B 0,C 180,E1 10666.858,E2 10666.858} C_VEL
LIN {X 0,Y 552.274,Z 717.248,A -85,B 0,C 180,E1 10667.472,E2 10667.472} C_VEL
LIN {X 0,Y 578.119,Z 765.932,A -85,B 0,C 180,E1 10670.504,E2 10670.504} C_VEL
LIN {X 0,Y 583.873,Z 780.43,A -85,B 0,C 180,E1 10671.277,E2 10671.277} C_VEL
LIN {X 0,Y 580.318,Z 824.765,A -85,B 0,C 180,E1 10672.453,E2 10672.453} C_VEL
LIN {X 0,Y 575.51,Z 868.807,A -85,B 0,C 180,E1 10674.262,E2 10674.262} C_VEL
LIN {X 0,Y 569.927,Z 911.937,A -85,B 0,C 180,E1 10676.785,E2 10676.785} C_VEL
LIN {X 0,Y 567.334,Z 930.006,A -85,B 0,C 180,E1 10678.111,E2 10678.111} C_VEL
LIN {X 0,Y 561.762,Z 943.895,A -85,B 0,C 180,E1 10679.047,E2 10679.047} C_VEL
LIN {X 0,Y 556.07,Z 957.209,A -85,B 0,C 180,E1 10680.056,E2 10680.056} C_VEL
LIN {X 0,Y 550.84,Z 990.676,A -85,B 0,C 180,E1 10683.708,E2 10683.708} C_VEL
LIN {X 0,Y 546.55,Z 1020.19,A -85,B 0,C 180,E1 10687.898,E2 10687.898} C_VEL
LIN {X 0,Y 543.516,Z 1044.898,A -85,B 0,C 180,E1 10692.558,E2 10692.558} C_VEL
LIN {X 0,Y 541.866,Z 1063.376,A -85,B 0,C 180,E1 10697.403,E2 10697.403} C_VEL
LIN {X 0,Y 541.204,Z 1074.948,A -85,B 0,C 180,E1 10701.951,E2 10701.951} C_VEL
LIN {X 0,Y 541.057,Z 1080.045,A -85,B 0,C 180,E1 10705.179,E2 10705.179} C_VEL
LIN {X 0,Y 541.098,Z 1082.953,A -85,B 0,C 180,E1 10709.999,E2 10709.999} C_VEL
LIN {X 0,Y 541.072,Z 1080.045,A -85,B 0,C 180,E1 10714.819,E2 10714.819} C_VEL
LIN {X 0,Y 541.251,Z 1073.348,A -85,B 0,C 180,E1 10718.857,E2 10718.857} C_VEL
LIN {X 0,Y 542.084,Z 1059.552,A -85,B 0,C 180,E1 10723.745,E2 10723.745} C_VEL
LIN {X 0,Y 543.931,Z 1040.618,A -85,B 0,C 180,E1 10728.333,E2 10728.333} C_VEL
LIN {X 0,Y 546.93,Z 1017.24,A -85,B 0,C 180,E1 10732.569,E2 10732.569} C_VEL
LIN {X 0,Y 551.465,Z 986.926,A -85,B 0,C 180,E1 10736.773,E2 10736.773} C_VEL
LIN {X 0,Y 557.411,Z 950.157,A -85,B 0,C 180,E1 10740.646,E2 10740.646} C_VEL
LIN {X 0,Y 563.639,Z 910.872,A -85,B 0,C 180,E1 10743.774,E2 10743.774} C_VEL
LIN {X 0,Y 569.674,Z 868.279,A -85,B 0,C 180,E1 10746.281,E2 10746.281} C_VEL
LIN {X 0,Y 574.705,Z 824.484,A -85,B 0,C 180,E1 10748.106,E2 10748.106} C_VEL
LIN {X 0,Y 577.613,Z 780.063,A -85,B 0,C 180,E1 10749.37,E2 10749.37} C_VEL
LIN {X 0,Y 558.319,Z 740.761,A -85,B 0,C 180,E1 10751.871,E2 10751.871} C_VEL
LIN {X 0,Y 539.779,Z 708.751,A -85,B 0,C 180,E1 10754.288,E2 10754.288} C_VEL
LIN {X 0,Y 539.627,Z 707.31,A -85,B 0,C 180,E1 10754.463,E2 10754.463} C_VEL
LIN {X 0,Y 539.623,Z 707.31,A -85,B 0,C 180,E1 10759.771,E2 10759.771} C_VEL
LIN {X 0,Y 539.752,Z 707.31,A -85,B 0,C 180,E1 10765.843,E2 10765.843} C_VEL
LIN {X 0,Y 539.855,Z 707.31,A -85,B 0,C 180,E1 10771.501,E2 10771.501} C_VEL
LIN {X 0,Y 539.848,Z 707.31,A -85,B 0,C 180,E1 10777.869,E2 10777.869} C_VEL
LIN {X 0,Y 540.065,Z 707.31,A -85,B 0,C 180,E1 10783.708,E2 10783.708} C_VEL
LIN {X 0,Y 540.457,Z 707.31,A -85,B 0,C 180,E1 10788.919,E2 10788.919} C_VEL
LIN {X 0,Y 540.534,Z 707.31,A -85,B 0,C 180,E1 10793.564,E2 10793.564} C_VEL
LIN {X 0,Y 540.578,Z 707.31,A -85,B 0,C 180,E1 10800.003,E2 10800.003} C_VEL
LIN {X 0,Y 540.342,Z 707.31,A -85,B 0,C 180,E1 10806.444,E2 10806.444} C_VEL
LIN {X 0,Y 540.26,Z 707.31,A -85,B 0,C 180,E1 10812.97,E2 10812.97} C_VEL
LIN {X 0,Y 540.055,Z 707.31,A -85,B 0,C 180,E1 10819.68,E2 10819.68} C_VEL
LIN {X 0,Y 539.87,Z 707.31,A -85,B 0,C 180,E1 10824.903,E2 10824.903} C_VEL
LIN {X 0,Y 539.693,Z 707.31,A -85,B 0,C 180,E1 10830.362,E2 10830.362} C_VEL
LIN {X 0,Y 539.656,Z 707.31,A -85,B 0,C 180,E1 10836.139,E2 10836.139} C_VEL
LIN {X 0,Y 539.668,Z 707.31,A -85,B 0,C 180,E1 10842.374,E2 10842.374} C_VEL
LIN {X 0,Y 539.726,Z 707.31,A -85,B 0,C 180,E1 10844.001,E2 10844.001} C_VEL
LIN {X 0,Y 542.451,Z 713.243,A -85,B 0,C 180,E1 10844.408,E2 10844.408} C_VEL
LIN {X 0,Y 566.675,Z 757.386,A -85,B 0,C 180,E1 10847.663,E2 10847.663} C_VEL
LIN {X 0,Y 576.751,Z 782.712,A -85,B 0,C 180,E1 10849.322,E2 10849.322} C_VEL
LIN {X 0,Y 572.23,Z 828.385,A -85,B 0,C 180,E1 10850.989,E2 10850.989} C_VEL
LIN {X 0,Y 566.259,Z 872.599,A -85,B 0,C 180,E1 10853.342,E2 10853.342} C_VEL
LIN {X 0,Y 560.091,Z 912.933,A -85,B 0,C 180,E1 10856.314,E2 10856.314} C_VEL
LIN {X 0,Y 553.644,Z 950.884,A -85,B 0,C 180,E1 10860.047,E2 10860.047} C_VEL
LIN {X 0,Y 548.463,Z 982.714,A -85,B 0,C 180,E1 10864.205,E2 10864.205} C_VEL
LIN {X 0,Y 544.715,Z 1009.152,A -85,B 0,C 180,E1 10868.799,E2 10868.799} C_VEL
LIN {X 0,Y 542.37,Z 1030.01,A -85,B 0,C 180,E1 10873.776,E2 10873.776} C_VEL
LIN {X 0,Y 541.369,Z 1043.894,A -85,B 0,C 180,E1 10878.701,E2 10878.701} C_VEL
LIN {X 0,Y 541.072,Z 1049.749,A -85,B 0,C 180,E1 10881.951,E2 10881.951} C_VEL
LIN {X 0,Y 540.876,Z 1053.836,A -85,B 0,C 180,E1 10886.788,E2 10886.788} C_VEL
LIN {X 0,Y 541.161,Z 1053.534,A -85,B 0,C 180,E1 10890.001,E2 10890.001} C_VEL
LIN {X 0,Y 541.15,Z 1048.474,A -85,B 0,C 180,E1 10894.82,E2 10894.82} C_VEL
LIN {X 0,Y 541.689,Z 1037.69,A -85,B 0,C 180,E1 10899.664,E2 10899.664} C_VEL
LIN {X 0,Y 543.07,Z 1022.441,A -85,B 0,C 180,E1 10904.133,E2 10904.133} C_VEL
LIN {X 0,Y 545.896,Z 1000.11,A -85,B 0,C 180,E1 10908.828,E2 10908.828} C_VEL
LIN {X 0,Y 550.236,Z 971.168,A -85,B 0,C 180,E1 10913.323,E2 10913.323} C_VEL
LIN {X 0,Y 555.84,Z 937.273,A -85,B 0,C 180,E1 10917.282,E2 10917.282} C_VEL
LIN {X 0,Y 562.124,Z 898.42,A -85,B 0,C 180,E1 10920.7,E2 10920.7} C_VEL
LIN {X 0,Y 568.321,Z 855.699,A -85,B 0,C 180,E1 10923.479,E2 10923.479} C_VEL
LIN {X 0,Y 573.54,Z 811.271,A -85,B 0,C 180,E1 10925.541,E2 10925.541} C_VEL
LIN {X 0,Y 575.796,Z 780.675,A -85,B 0,C 180,E1 10926.588,E2 10926.588} C_VEL
LIN {X 0,Y 556.422,Z 738.472,A -85,B 0,C 180,E1 10929.351,E2 10929.351} C_VEL
LIN {X 0,Y 539.877,Z 708.836,A -85,B 0,C 180,E1 10931.435,E2 10931.435} C_VEL
LIN {X 0,Y 539.721,Z 707.31,A -85,B 0,C 180,E1 10931.58,E2 10931.58} C_VEL
LIN {X 0,Y 539.677,Z 707.31,A -85,B 0,C 180,E1 10937.627,E2 10937.627} C_VEL
LIN {X 0,Y 539.696,Z 707.31,A -85,B 0,C 180,E1 10943.864,E2 10943.864} C_VEL
LIN {X 0,Y 539.837,Z 707.31,A -85,B 0,C 180,E1 10949.647,E2 10949.647} C_VEL
LIN {X 0,Y 539.85,Z 707.31,A -85,B 0,C 180,E1 10955.096,E2 10955.096} C_VEL
LIN {X 0,Y 539.978,Z 707.31,A -85,B 0,C 180,E1 10960.317,E2 10960.317} C_VEL
LIN {X 0,Y 540.423,Z 707.31,A -85,B 0,C 180,E1 10967.034,E2 10967.034} C_VEL
LIN {X 0,Y 540.582,Z 707.31,A -85,B 0,C 180,E1 10971.94,E2 10971.94} C_VEL
LIN {X 0,Y 540.403,Z 707.31,A -85,B 0,C 180,E1 10976.782,E2 10976.782} C_VEL
LIN {X 0,Y 540.714,Z 707.31,A -85,B 0,C 180,E1 10981.603,E2 10981.603} C_VEL
LIN {X 0,Y 540.627,Z 707.31,A -85,B 0,C 180,E1 10988.054,E2 10988.054} C_VEL
LIN {X 0,Y 540.3,Z 707.31,A -85,B 0,C 180,E1 10992.963,E2 10992.963} C_VEL
LIN {X 0,Y 540.01,Z 707.31,A -85,B 0,C 180,E1 10997.977,E2 10997.977} C_VEL
LIN {X 0,Y 539.88,Z 707.31,A -85,B 0,C 180,E1 11003.136,E2 11003.136} C_VEL
LIN {X 0,Y 539.856,Z 707.31,A -85,B 0,C 180,E1 11008.499,E2 11008.499} C_VEL
LIN {X 0,Y 539.759,Z 707.31,A -85,B 0,C 180,E1 11014.156,E2 11014.156} C_VEL
LIN {X 0,Y 539.642,Z 707.31,A -85,B 0,C 180,E1 11020.693,E2 11020.693} C_VEL
LIN {X 0,Y 539.67,Z 707.746,A -85,B 0,C 180,E1 11026.107,E2 11026.107} C_VEL
LIN {X 0,Y 545.29,Z 718.468,A -85,B 0,C 180,E1 11026.84,E2 11026.84} C_VEL
LIN {X 0,Y 572.114,Z 769.281,A -85,B 0,C 180,E1 11030.087,E2 11030.087} C_VEL
LIN {X 0,Y 577.458,Z 783.055,A -85,B 0,C 180,E1 11030.847,E2 11030.847} C_VEL
LIN {X 0,Y 573.662,Z 827.975,A -85,B 0,C 180,E1 11032.097,E2 11032.097} C_VEL
LIN {X 0,Y 568.733,Z 870.305,A -85,B 0,C 180,E1 11033.886,E2 11033.886} C_VEL
LIN {X 0,Y 563.013,Z 912.284,A -85,B 0,C 180,E1 11036.38,E2 11036.38} C_VEL
LIN {X 0,Y 556.795,Z 953.004,A -85,B 0,C 180,E1 11039.654,E2 11039.654} C_VEL
LIN {X 0,Y 556.07,Z 957.209,A -85,B 0,C 180,E1 11040.056,E2 11040.056} C_VEL
LIN {X 0,Y 550.473,Z 970.02,A -85,B 0,C 180,E1 11041.159,E2 11041.159} C_VEL
LIN {X 0,Y 544.85,Z 982.212,A -85,B 0,C 180,E1 11042.335,E2 11042.335} C_VEL
LIN {X 0,Y 540.091,Z 1012.161,A -85,B 0,C 180,E1 11046.343,E2 11046.343} C_VEL
LIN {X 0,Y 536.489,Z 1038.287,A -85,B 0,C 180,E1 11050.94,E2 11050.94} C_VEL
LIN {X 0,Y 534.455,Z 1057.963,A -85,B 0,C 180,E1 11055.634,E2 11055.634} C_VEL
LIN {X 0,Y 533.517,Z 1071.203,A -85,B 0,C 180,E1 11060.187,E2 11060.187} C_VEL
LIN {X 0,Y 533.246,Z 1078.45,A -85,B 0,C 180,E1 11064.032,E2 11064.032} C_VEL
LIN {X 0,Y 533.072,Z 1082.397,A -85,B 0,C 180,E1 11068.37,E2 11068.37} C_VEL
LIN {X 0,Y 533.204,Z 1081.429,A -85,B 0,C 180,E1 11073.258,E2 11073.258} C_VEL
LIN {X 0,Y 533.283,Z 1074.73,A -85,B 0,C 180,E1 11078.168,E2 11078.168} C_VEL
LIN {X 0,Y 533.952,Z 1063.962,A -85,B 0,C 180,E1 11082.531,E2 11082.531} C_VEL
LIN {X 0,Y 535.552,Z 1046.427,A -85,B 0,C 180,E1 11087.283,E2 11087.283} C_VEL
LIN {X 0,Y 538.321,Z 1024.015,A -85,B 0,C 180,E1 11091.736,E2 11091.736} C_VEL
LIN {X 0,Y 542.507,Z 996.776,A -85,B 0,C 180,E1 11095.877,E2 11095.877} C_VEL
LIN {X 0,Y 548.267,Z 962.841,A -85,B 0,C 180,E1 11099.835,E2 11099.835} C_VEL
LIN {X 0,Y 554.829,Z 923.947,A -85,B 0,C 180,E1 11103.276,E2 11103.276} C_VEL
LIN {X 0,Y 561.354,Z 881.425,A -85,B 0,C 180,E1 11106.074,E2 11106.074} C_VEL
LIN {X 0,Y 567.269,Z 835.56,A -85,B 0,C 180,E1 11108.213,E2 11108.213} C_VEL
LIN {X 0,Y 571.791,Z 786.283,A -85,B 0,C 180,E1 11109.699,E2 11109.699} C_VEL
LIN {X 0,Y 569.288,Z 777.762,A -85,B 0,C 180,E1 11110.131,E2 11110.131} C_VEL
LIN {X 0,Y 548.869,Z 737.713,A -85,B 0,C 180,E1 11112.835,E2 11112.835} C_VEL
LIN {X 0,Y 531.796,Z 708.447,A -85,B 0,C 180,E1 11115.159,E2 11115.159} C_VEL
LIN {X 0,Y 531.708,Z 707.31,A -85,B 0,C 180,E1 11115.265,E2 11115.265} C_VEL
LIN {X 0,Y 531.703,Z 707.31,A -85,B 0,C 180,E1 11121.174,E2 11121.174} C_VEL
LIN {X 0,Y 531.88,Z 707.31,A -85,B 0,C 180,E1 11127.229,E2 11127.229} C_VEL
LIN {X 0,Y 531.924,Z 707.31,A -85,B 0,C 180,E1 11132.886,E2 11132.886} C_VEL
LIN {X 0,Y 531.95,Z 707.31,A -85,B 0,C 180,E1 11138.267,E2 11138.267} C_VEL
LIN {X 0,Y 532.146,Z 707.31,A -85,B 0,C 180,E1 11143.458,E2 11143.458} C_VEL
LIN {X 0,Y 532.501,Z 707.31,A -85,B 0,C 180,E1 11148.513,E2 11148.513} C_VEL
LIN {X 0,Y 532.64,Z 707.31,A -85,B 0,C 180,E1 11153.468,E2 11153.468} C_VEL
LIN {X 0,Y 532.674,Z 707.31,A -85,B 0,C 180,E1 11160.003,E2 11160.003} C_VEL
LIN {X 0,Y 532.422,Z 707.31,A -85,B 0,C 180,E1 11166.54,E2 11166.54} C_VEL
LIN {X 0,Y 532.328,Z 707.31,A -85,B 0,C 180,E1 11173.167,E2 11173.167} C_VEL
LIN {X 0,Y 532.12,Z 707.31,A -85,B 0,C 180,E1 11179.986,E2 11179.986} C_VEL
LIN {X 0,Y 531.924,Z 707.31,A -85,B 0,C 180,E1 11185.301,E2 11185.301} C_VEL
LIN {X 0,Y 531.72,Z 707.31,A -85,B 0,C 180,E1 11191.242,E2 11191.242} C_VEL
LIN {X 0,Y 531.711,Z 707.31,A -85,B 0,C 180,E1 11197.061,E2 11197.061} C_VEL
LIN {X 0,Y 531.769,Z 707.582,A -85,B 0,C 180,E1 11203.155,E2 11203.155} C_VEL
LIN {X 0,Y 534.566,Z 713.324,A -85,B 0,C 180,E1 11203.571,E2 11203.571} C_VEL
LIN {X 0,Y 559.371,Z 757.819,A -85,B 0,C 180,E1 11207.012,E2 11207.012} C_VEL
LIN {X 0,Y 570.463,Z 784.952,A -85,B 0,C 180,E1 11208.878,E2 11208.878} C_VEL
LIN {X 0,Y 565.805,Z 829.677,A -85,B 0,C 180,E1 11210.546,E2 11210.546} C_VEL
LIN {X 0,Y 559.751,Z 872.674,A -85,B 0,C 180,E1 11212.858,E2 11212.858} C_VEL
LIN {X 0,Y 553.117,Z 914.086,A -85,B 0,C 180,E1 11215.95,E2 11215.95} C_VEL
LIN {X 0,Y 546.665,Z 950.522,A -85,B 0,C 180,E1 11219.575,E2 11219.575} C_VEL
LIN {X 0,Y 541.161,Z 982.311,A -85,B 0,C 180,E1 11223.76,E2 11223.76} C_VEL
LIN {X 0,Y 537.098,Z 1009.216,A -85,B 0,C 180,E1 11228.483,E2 11228.483} C_VEL
LIN {X 0,Y 534.591,Z 1030.111,A -85,B 0,C 180,E1 11233.533,E2 11233.533} C_VEL
LIN {X 0,Y 533.518,Z 1044.036,A -85,B 0,C 180,E1 11238.532,E2 11238.532} C_VEL
LIN {X 0,Y 533.204,Z 1049.917,A -85,B 0,C 180,E1 11241.831,E2 11241.831} C_VEL
LIN {X 0,Y 533.04,Z 1053.275,A -85,B 0,C 180,E1 11245.108,E2 11245.108} C_VEL
LIN {X 0,Y 533.261,Z 1053.764,A -85,B 0,C 180,E1 11250.001,E2 11250.001} C_VEL
LIN {X 0,Y 533.265,Z 1048.729,A -85,B 0,C 180,E1 11254.891,E2 11254.891} C_VEL
LIN {X 0,Y 533.858,Z 1037.987,A -85,B 0,C 180,E1 11259.807,E2 11259.807} C_VEL
LIN {X 0,Y 535.343,Z 1022.782,A -85,B 0,C 180,E1 11264.341,E2 11264.341} C_VEL
LIN {X 0,Y 538.254,Z 1000.838,A -85,B 0,C 180,E1 11269.041,E2 11269.041} C_VEL
LIN {X 0,Y 542.88,Z 971.564,A -85,B 0,C 180,E1 11273.658,E2 11273.658} C_VEL
LIN {X 0,Y 548.814,Z 937.364,A -85,B 0,C 180,E1 11277.698,E2 11277.698} C_VEL
LIN {X 0,Y 555.297,Z 898.911,A -85,B 0,C 180,E1 11281.119,E2 11281.119} C_VEL
LIN {X 0,Y 561.729,Z 856.292,A -85,B 0,C 180,E1 11283.924,E2 11283.924} C_VEL
LIN {X 0,Y 567.167,Z 811.944,A -85,B 0,C 180,E1 11286.003,E2 11286.003} C_VEL
LIN {X 0,Y 569.308,Z 783.387,A -85,B 0,C 180,E1 11287.005,E2 11287.005} C_VEL
LIN {X 0,Y 550.849,Z 742.52,A -85,B 0,C 180,E1 11289.772,E2 11289.772} C_VEL
LIN {X 0,Y 531.81,Z 708.328,A -85,B 0,C 180,E1 11292.255,E2 11292.255} C_VEL
LIN {X 0,Y 531.734,Z 707.31,A -85,B 0,C 180,E1 11292.641,E2 11292.641} C_VEL
LIN {X 0,Y 531.756,Z 707.31,A -85,B 0,C 180,E1 11299.043,E2 11299.043} C_VEL
LIN {X 0,Y 531.837,Z 707.31,A -85,B 0,C 180,E1 11305.723,E2 11305.723} C_VEL
LIN {X 0,Y 531.886,Z 707.31,A -85,B 0,C 180,E1 11312.035,E2 11312.035} C_VEL
LIN {X 0,Y 532.006,Z 707.31,A -85,B 0,C 180,E1 11318.263,E2 11318.263} C_VEL
LIN {X 0,Y 532.195,Z 707.31,A -85,B 0,C 180,E1 11323.454,E2 11323.454} C_VEL
LIN {X 0,Y 532.605,Z 707.31,A -85,B 0,C 180,E1 11328.509,E2 11328.509} C_VEL
LIN {X 0,Y 532.72,Z 707.31,A -85,B 0,C 180,E1 11334.646,E2 11334.646} C_VEL
LIN {X 0,Y 532.801,Z 707.31,A -85,B 0,C 180,E1 11341.627,E2 11341.627} C_VEL
LIN {X 0,Y 532.722,Z 707.31,A -85,B 0,C 180,E1 11348.174,E2 11348.174} C_VEL
LIN {X 0,Y 532.325,Z 707.31,A -85,B 0,C 180,E1 11354.555,E2 11354.555} C_VEL
LIN {X 0,Y 532.023,Z 707.31,A -85,B 0,C 180,E1 11359.983,E2 11359.983} C_VEL
LIN {X 0,Y 531.925,Z 707.31,A -85,B 0,C 180,E1 11365.295,E2 11365.295} C_VEL
LIN {X 0,Y 531.869,Z 707.31,A -85,B 0,C 180,E1 11371.266,E2 11371.266} C_VEL
LIN {X 0,Y 531.732,Z 707.31,A -85,B 0,C 180,E1 11377.061,E2 11377.061} C_VEL
LIN {X 0,Y 531.707,Z 707.31,A -85,B 0,C 180,E1 11383.153,E2 11383.153} C_VEL
LIN {X 0,Y 531.741,Z 707.995,A -85,B 0,C 180,E1 11385.314,E2 11385.314} C_VEL
LIN {X 0,Y 561.227,Z 762.495,A -85,B 0,C 180,E1 11389.051,E2 11389.051} C_VEL
LIN {X 0,Y 571.136,Z 785.161,A -85,B 0,C 180,E1 11390.399,E2 11390.399} C_VEL
LIN {X 0,Y 566.986,Z 831.53,A -85,B 0,C 180,E1 11391.746,E2 11391.746} C_VEL
LIN {X 0,Y 561.546,Z 875.491,A -85,B 0,C 180,E1 11393.699,E2 11393.699} C_VEL
LIN {X 0,Y 555.536,Z 916.539,A -85,B 0,C 180,E1 11396.251,E2 11396.251} C_VEL
LIN {X 0,Y 549.385,Z 954.821,A -85,B 0,C 180,E1 11399.43,E2 11399.43} C_VEL
LIN {X 0,Y 544.85,Z 982.212,A -85,B 0,C 180,E1 11402.335,E2 11402.335} C_VEL
LIN {X 0,Y 539.261,Z 993.837,A -85,B 0,C 180,E1 11403.596,E2 11403.596} C_VEL
LIN {X 0,Y 533.782,Z 1004.8,A -85,B 0,C 180,E1 11404.932,E2 11404.932} C_VEL
LIN {X 0,Y 529.711,Z 1031.035,A -85,B 0,C 180,E1 11409.266,E2 11409.266} C_VEL
LIN {X 0,Y 527.194,Z 1051.58,A -85,B 0,C 180,E1 11413.743,E2 11413.743} C_VEL
LIN {X 0,Y 525.851,Z 1068.071,A -85,B 0,C 180,E1 11418.829,E2 11418.829} C_VEL
LIN {X 0,Y 525.341,Z 1077.397,A -85,B 0,C 180,E1 11423.373,E2 11423.373} C_VEL
LIN {X 0,Y 525.201,Z 1082.187,A -85,B 0,C 180,E1 11428.346,E2 11428.346} C_VEL
LIN {X 0,Y 525.381,Z 1082.191,A -85,B 0,C 180,E1 11431.652,E2 11431.652} C_VEL
LIN {X 0,Y 525.3,Z 1077.391,A -85,B 0,C 180,E1 11436.626,E2 11436.626} C_VEL
LIN {X 0,Y 525.818,Z 1068.063,A -85,B 0,C 180,E1 11441.169,E2 11441.169} C_VEL
LIN {X 0,Y 527.288,Z 1051.493,A -85,B 0,C 180,E1 11446.273,E2 11446.273} C_VEL
LIN {X 0,Y 530.207,Z 1027.777,A -85,B 0,C 180,E1 11451.371,E2 11451.371} C_VEL
LIN {X 0,Y 534.905,Z 998.237,A -85,B 0,C 180,E1 11456.047,E2 11456.047} C_VEL
LIN {X 0,Y 541.227,Z 962.725,A -85,B 0,C 180,E1 11460.263,E2 11460.263} C_VEL
LIN {X 0,Y 548.093,Z 923.846,A -85,B 0,C 180,E1 11463.742,E2 11463.742} C_VEL
LIN {X 0,Y 555.009,Z 880.779,A -85,B 0,C 180,E1 11466.594,E2 11466.594} C_VEL
LIN {X 0,Y 560.97,Z 836.216,A -85,B 0,C 180,E1 11468.69,E2 11468.69} C_VEL
LIN {X 0,Y 565.597,Z 788.123,A -85,B 0,C 180,E1 11470.171,E2 11470.171} C_VEL
LIN {X 0,Y 553.387,Z 759.879,A -85,B 0,C 180,E1 11471.984,E2 11471.984} C_VEL
LIN {X 0,Y 529.575,Z 718.529,A -85,B 0,C 180,E1 11475.214,E2 11475.214} C_VEL
LIN {X 0,Y 523.796,Z 708.06,A -85,B 0,C 180,E1 11476.074,E2 11476.074} C_VEL
LIN {X 0,Y 523.781,Z 707.31,A -85,B 0,C 180,E1 11481.366,E2 11481.366} C_VEL
LIN {X 0,Y 523.961,Z 707.31,A -85,B 0,C 180,E1 11487.006,E2 11487.006} C_VEL
LIN {X 0,Y 524.024,Z 707.31,A -85,B 0,C 180,E1 11492.443,E2 11492.443} C_VEL
LIN {X 0,Y 524.005,Z 707.31,A -85,B 0,C 180,E1 11497.92,E2 11497.92} C_VEL
LIN {X 0,Y 524.203,Z 707.31,A -85,B 0,C 180,E1 11503.2,E2 11503.2} C_VEL
LIN {X 0,Y 524.601,Z 707.31,A -85,B 0,C 180,E1 11509.153,E2 11509.153} C_VEL
LIN {X 0,Y 524.732,Z 707.31,A -85,B 0,C 180,E1 11513.37,E2 11513.37} C_VEL
LIN {X 0,Y 524.771,Z 707.31,A -85,B 0,C 180,E1 11520.003,E2 11520.003} C_VEL
LIN {X 0,Y 524.499,Z 707.31,A -85,B 0,C 180,E1 11526.639,E2 11526.639} C_VEL
LIN {X 0,Y 524.504,Z 707.31,A -85,B 0,C 180,E1 11531.671,E2 11531.671} C_VEL
LIN {X 0,Y 524.181,Z 707.31,A -85,B 0,C 180,E1 11537.444,E2 11537.444} C_VEL
LIN {X 0,Y 524.116,Z 707.31,A -85,B 0,C 180,E1 11543.881,E2 11543.881} C_VEL
LIN {X 0,Y 523.798,Z 707.31,A -85,B 0,C 180,E1 11549.783,E2 11549.783} C_VEL
LIN {X 0,Y 523.752,Z 707.31,A -85,B 0,C 180,E1 11555.892,E2 11555.892} C_VEL
LIN {X 0,Y 523.873,Z 707.683,A -85,B 0,C 180,E1 11562.261,E2 11562.261} C_VEL
LIN {X 0,Y 526.669,Z 713.35,A -85,B 0,C 180,E1 11562.693,E2 11562.693} C_VEL
LIN {X 0,Y 550.867,Z 756.102,A -85,B 0,C 180,E1 11566.163,E2 11566.163} C_VEL
LIN {X 0,Y 564.169,Z 787.895,A -85,B 0,C 180,E1 11568.448,E2 11568.448} C_VEL
LIN {X 0,Y 559.348,Z 831.47,A -85,B 0,C 180,E1 11570.116,E2 11570.116} C_VEL
LIN {X 0,Y 553.147,Z 873.545,A -85,B 0,C 180,E1 11572.415,E2 11572.415} C_VEL
LIN {X 0,Y 546.39,Z 913.952,A -85,B 0,C 180,E1 11575.459,E2 11575.459} C_VEL
LIN {X 0,Y 539.512,Z 951.235,A -85,B 0,C 180,E1 11579.217,E2 11579.217} C_VEL
LIN {X 0,Y 533.624,Z 983.481,A -85,B 0,C 180,E1 11583.54,E2 11583.54} C_VEL
LIN {X 0,Y 529.303,Z 1010.67,A -85,B 0,C 180,E1 11588.447,E2 11588.447} C_VEL
LIN {X 0,Y 526.835,Z 1030.214,A -85,B 0,C 180,E1 11593.284,E2 11593.284} C_VEL
LIN {X 0,Y 525.677,Z 1044.178,A -85,B 0,C 180,E1 11598.359,E2 11598.359} C_VEL
LIN {X 0,Y 525.223,Z 1051.238,A -85,B 0,C 180,E1 11602.541,E2 11602.541} C_VEL
LIN {X 0,Y 525.084,Z 1054.245,A -85,B 0,C 180,E1 11606.692,E2 11606.692} C_VEL
LIN {X 0,Y 525.372,Z 1053.993,A -85,B 0,C 180,E1 11610.001,E2 11610.001} C_VEL
LIN {X 0,Y 525.39,Z 1048.984,A -85,B 0,C 180,E1 11614.965,E2 11614.965} C_VEL
LIN {X 0,Y 526.027,Z 1038.283,A -85,B 0,C 180,E1 11619.954,E2 11619.954} C_VEL
LIN {X 0,Y 527.617,Z 1023.114,A -85,B 0,C 180,E1 11624.556,E2 11624.556} C_VEL
LIN {X 0,Y 530.808,Z 1000.412,A -85,B 0,C 180,E1 11629.462,E2 11629.462} C_VEL
LIN {X 0,Y 535.566,Z 971.95,A -85,B 0,C 180,E1 11634.001,E2 11634.001} C_VEL
LIN {X 0,Y 541.667,Z 938.309,A -85,B 0,C 180,E1 11638.039,E2 11638.039} C_VEL
LIN {X 0,Y 548.432,Z 899.814,A -85,B 0,C 180,E1 11641.517,E2 11641.517} C_VEL
LIN {X 0,Y 555.184,Z 856.855,A -85,B 0,C 180,E1 11644.38,E2 11644.38} C_VEL
LIN {X 0,Y 560.961,Z 811.322,A -85,B 0,C 180,E1 11646.529,E2 11646.529} C_VEL
LIN {X 0,Y 562.885,Z 786.192,A -85,B 0,C 180,E1 11647.425,E2 11647.425} C_VEL
LIN {X 0,Y 544.68,Z 745.431,A -85,B 0,C 180,E1 11650.283,E2 11650.283} C_VEL
LIN {X 0,Y 523.865,Z 708.027,A -85,B 0,C 180,E1 11653.095,E2 11653.095} C_VEL
LIN {X 0,Y 523.859,Z 707.31,A -85,B 0,C 180,E1 11658.775,E2 11658.775} C_VEL
LIN {X 0,Y 523.809,Z 707.31,A -85,B 0,C 180,E1 11664.644,E2 11664.644} C_VEL
LIN {X 0,Y 523.944,Z 707.31,A -85,B 0,C 180,E1 11670.545,E2 11670.545} C_VEL
LIN {X 0,Y 524.05,Z 707.31,A -85,B 0,C 180,E1 11676.116,E2 11676.116} C_VEL
LIN {X 0,Y 524.206,Z 707.31,A -85,B 0,C 180,E1 11682.552,E2 11682.552} C_VEL
LIN {X 0,Y 524.69,Z 707.31,A -85,B 0,C 180,E1 11688.333,E2 11688.333} C_VEL
LIN {X 0,Y 524.813,Z 707.31,A -85,B 0,C 180,E1 11693.365,E2 11693.365} C_VEL
LIN {X 0,Y 524.79,Z 707.31,A -85,B 0,C 180,E1 11699.997,E2 11699.997} C_VEL
LIN {X 0,Y 524.746,Z 707.31,A -85,B 0,C 180,E1 11706.63,E2 11706.63} C_VEL
LIN {X 0,Y 524.587,Z 707.31,A -85,B 0,C 180,E1 11711.663,E2 11711.663} C_VEL
LIN {X 0,Y 524.16,Z 707.31,A -85,B 0,C 180,E1 11717.432,E2 11717.432} C_VEL
LIN {X 0,Y 524.026,Z 707.31,A -85,B 0,C 180,E1 11723.879,E2 11723.879} C_VEL
LIN {X 0,Y 523.951,Z 707.31,A -85,B 0,C 180,E1 11729.809,E2 11729.809} C_VEL
LIN {X 0,Y 523.816,Z 707.31,A -85,B 0,C 180,E1 11735.899,E2 11735.899} C_VEL
LIN {X 0,Y 523.804,Z 707.31,A -85,B 0,C 180,E1 11741.709,E2 11741.709} C_VEL
LIN {X 0,Y 523.788,Z 707.31,A -85,B 0,C 180,E1 11744.464,E2 11744.464} C_VEL
LIN {X 0,Y 526.417,Z 713.186,A -85,B 0,C 180,E1 11744.855,E2 11744.855} C_VEL
LIN {X 0,Y 553.071,Z 761.327,A -85,B 0,C 180,E1 11748.317,E2 11748.317} C_VEL
LIN {X 0,Y 564.748,Z 788.05,A -85,B 0,C 180,E1 11749.967,E2 11749.967} C_VEL
LIN {X 0,Y 560.529,Z 832.877,A -85,B 0,C 180,E1 11751.305,E2 11751.305} C_VEL
LIN {X 0,Y 554.574,Z 878.899,A -85,B 0,C 180,E1 11753.411,E2 11753.411} C_VEL
LIN {X 0,Y 547.95,Z 921.549,A -85,B 0,C 180,E1 11756.175,E2 11756.175} C_VEL
LIN {X 0,Y 541.381,Z 959.982,A -85,B 0,C 180,E1 11759.529,E2 11759.529} C_VEL
LIN {X 0,Y 535.703,Z 993.036,A -85,B 0,C 180,E1 11763.315,E2 11763.315} C_VEL
LIN {X 0,Y 533.782,Z 1004.8,A -85,B 0,C 180,E1 11764.932,E2 11764.932} C_VEL
LIN {X 0,Y 528.363,Z 1015.131,A -85,B 0,C 180,E1 11766.347,E2 11766.347} C_VEL
LIN {X 0,Y 523.031,Z 1024.776,A -85,B 0,C 180,E1 11767.834,E2 11767.834} C_VEL
LIN {X 0,Y 519.867,Z 1047.75,A -85,B 0,C 180,E1 11772.615,E2 11772.615} C_VEL
LIN {X 0,Y 518.228,Z 1064.223,A -85,B 0,C 180,E1 11777.33,E2 11777.33} C_VEL
LIN {X 0,Y 517.518,Z 1075.904,A -85,B 0,C 180,E1 11782.427,E2 11782.427} C_VEL
LIN {X 0,Y 517.328,Z 1081.007,A -85,B 0,C 180,E1 11786.641,E2 11786.641} C_VEL
LIN {X 0,Y 517.478,Z 1081.979,A -85,B 0,C 180,E1 11791.677,E2 11791.677} C_VEL
LIN {X 0,Y 517.418,Z 1077.178,A -85,B 0,C 180,E1 11796.727,E2 11796.727} C_VEL
LIN {X 0,Y 517.947,Z 1067.877,A -85,B 0,C 180,E1 11801.331,E2 11801.331} C_VEL
LIN {X 0,Y 519.521,Z 1051.074,A -85,B 0,C 180,E1 11806.581,E2 11806.581} C_VEL
LIN {X 0,Y 522.512,Z 1028.286,A -85,B 0,C 180,E1 11811.566,E2 11811.566} C_VEL
LIN {X 0,Y 527.569,Z 998.092,A -85,B 0,C 180,E1 11816.437,E2 11816.437} C_VEL
LIN {X 0,Y 534.235,Z 962.615,A -85,B 0,C 180,E1 11820.702,E2 11820.702} C_VEL
LIN {X 0,Y 541.404,Z 923.778,A -85,B 0,C 180,E1 11824.216,E2 11824.216} C_VEL
LIN {X 0,Y 548.588,Z 880.836,A -85,B 0,C 180,E1 11827.089,E2 11827.089} C_VEL
LIN {X 0,Y 554.944,Z 835.095,A -85,B 0,C 180,E1 11829.252,E2 11829.252} C_VEL
LIN {X 0,Y 558.894,Z 788.047,A -85,B 0,C 180,E1 11830.764,E2 11830.764} C_VEL
LIN {X 0,Y 540.65,Z 750.085,A -85,B 0,C 180,E1 11833.442,E2 11833.442} C_VEL
LIN {X 0,Y 517.441,Z 712.086,A -85,B 0,C 180,E1 11836.747,E2 11836.747} C_VEL
LIN {X 0,Y 515.817,Z 707.31,A -85,B 0,C 180,E1 11837.091,E2 11837.091} C_VEL
LIN {X 0,Y 515.901,Z 707.31,A -85,B 0,C 180,E1 11842.474,E2 11842.474} C_VEL
LIN {X 0,Y 516.053,Z 707.31,A -85,B 0,C 180,E1 11848.383,E2 11848.383} C_VEL
LIN {X 0,Y 516.068,Z 707.31,A -85,B 0,C 180,E1 11853.87,E2 11853.87} C_VEL
LIN {X 0,Y 516.144,Z 707.31,A -85,B 0,C 180,E1 11859.969,E2 11859.969} C_VEL
LIN {X 0,Y 516.491,Z 707.31,A -85,B 0,C 180,E1 11866.428,E2 11866.428} C_VEL
LIN {X 0,Y 516.857,Z 707.31,A -85,B 0,C 180,E1 11871.573,E2 11871.573} C_VEL
LIN {X 0,Y 516.978,Z 707.31,A -85,B 0,C 180,E1 11878.323,E2 11878.323} C_VEL
LIN {X 0,Y 516.772,Z 707.31,A -85,B 0,C 180,E1 11885.05,E2 11885.05} C_VEL
LIN {X 0,Y 516.571,Z 707.31,A -85,B 0,C 180,E1 11891.853,E2 11891.853} C_VEL
LIN {X 0,Y 516.295,Z 707.31,A -85,B 0,C 180,E1 11897.071,E2 11897.071} C_VEL
LIN {X 0,Y 516.246,Z 707.31,A -85,B 0,C 180,E1 11902.436,E2 11902.436} C_VEL
LIN {X 0,Y 515.938,Z 707.31,A -85,B 0,C 180,E1 11908.22,E2 11908.22} C_VEL
LIN {X 0,Y 515.814,Z 707.31,A -85,B 0,C 180,E1 11913.934,E2 11913.934} C_VEL
LIN {X 0,Y 515.873,Z 707.31,A -85,B 0,C 180,E1 11920.264,E2 11920.264} C_VEL
LIN {X 0,Y 515.97,Z 707.31,A -85,B 0,C 180,E1 11921.3,E2 11921.3} C_VEL
LIN {X 0,Y 518.546,Z 713.168,A -85,B 0,C 180,E1 11921.741,E2 11921.741} C_VEL
LIN {X 0,Y 542.525,Z 754.378,A -85,B 0,C 180,E1 11925.289,E2 11925.289} C_VEL
LIN {X 0,Y 557.938,Z 789.875,A -85,B 0,C 180,E1 11927.972,E2 11927.972} C_VEL
LIN {X 0,Y 552.946,Z 833.147,A -85,B 0,C 180,E1 11929.672,E2 11929.672} C_VEL
LIN {X 0,Y 546.695,Z 873.82,A -85,B 0,C 180,E1 11931.921,E2 11931.921} C_VEL
LIN {X 0,Y 539.573,Z 914.577,A -85,B 0,C 180,E1 11935.027,E2 11935.027} C_VEL
LIN {X 0,Y 532.573,Z 950.993,A -85,B 0,C 180,E1 11938.735,E2 11938.735} C_VEL
LIN {X 0,Y 526.245,Z 984.008,A -85,B 0,C 180,E1 11943.218,E2 11943.218} C_VEL
LIN {X 0,Y 521.975,Z 1009.392,A -85,B 0,C 180,E1 11947.827,E2 11947.827} C_VEL
LIN {X 0,Y 519.098,Z 1030.331,A -85,B 0,C 180,E1 11953.027,E2 11953.027} C_VEL
LIN {X 0,Y 517.815,Z 1044.321,A -85,B 0,C 180,E1 11958.18,E2 11958.18} C_VEL
LIN {X 0,Y 517.337,Z 1051.418,A -85,B 0,C 180,E1 11962.426,E2 11962.426} C_VEL
LIN {X 0,Y 517.183,Z 1054.45,A -85,B 0,C 180,E1 11966.641,E2 11966.641} C_VEL
LIN {X 0,Y 517.472,Z 1054.223,A -85,B 0,C 180,E1 11970.001,E2 11970.001} C_VEL
LIN {X 0,Y 517.534,Z 1048.765,A -85,B 0,C 180,E1 11975.376,E2 11975.376} C_VEL
LIN {X 0,Y 518.356,Z 1037.449,A -85,B 0,C 180,E1 11980.529,E2 11980.529} C_VEL
LIN {X 0,Y 520.136,Z 1021.729,A -85,B 0,C 180,E1 11985.202,E2 11985.202} C_VEL
LIN {X 0,Y 523.426,Z 999.805,A -85,B 0,C 180,E1 11989.926,E2 11989.926} C_VEL
LIN {X 0,Y 528.258,Z 972.331,A -85,B 0,C 180,E1 11994.355,E2 11994.355} C_VEL
LIN {X 0,Y 534.457,Z 939.555,A -85,B 0,C 180,E1 11998.355,E2 11998.355} C_VEL
LIN {X 0,Y 541.699,Z 899.951,A -85,B 0,C 180,E1 12001.985,E2 12001.985} C_VEL
LIN {X 0,Y 548.667,Z 857.411,A -85,B 0,C 180,E1 12004.847,E2 12004.847} C_VEL
LIN {X 0,Y 554.487,Z 813.273,A -85,B 0,C 180,E1 12006.961,E2 12006.961} C_VEL
LIN {X 0,Y 556.39,Z 788.621,A -85,B 0,C 180,E1 12007.878,E2 12007.878} C_VEL
LIN {X 0,Y 538.601,Z 748.415,A -85,B 0,C 180,E1 12010.791,E2 12010.791} C_VEL
LIN {X 0,Y 516.016,Z 708.676,A -85,B 0,C 180,E1 12013.944,E2 12013.944} C_VEL
LIN {X 0,Y 515.894,Z 707.31,A -85,B 0,C 180,E1 12013.988,E2 12013.988} C_VEL
LIN {X 0,Y 515.884,Z 707.31,A -85,B 0,C 180,E1 12019.797,E2 12019.797} C_VEL
LIN {X 0,Y 515.928,Z 707.31,A -85,B 0,C 180,E1 12026.074,E2 12026.074} C_VEL
LIN {X 0,Y 516.043,Z 707.31,A -85,B 0,C 180,E1 12031.972,E2 12031.972} C_VEL
LIN {X 0,Y 516.148,Z 707.31,A -85,B 0,C 180,E1 12037.559,E2 12037.559} C_VEL
LIN {X 0,Y 516.335,Z 707.31,A -85,B 0,C 180,E1 12042.93,E2 12042.93} C_VEL
LIN {X 0,Y 516.757,Z 707.31,A -85,B 0,C 180,E1 12048.151,E2 12048.151} C_VEL
LIN {X 0,Y 516.914,Z 707.31,A -85,B 0,C 180,E1 12053.263,E2 12053.263} C_VEL
LIN {X 0,Y 516.887,Z 707.31,A -85,B 0,C 180,E1 12059.997,E2 12059.997} C_VEL
LIN {X 0,Y 516.861,Z 707.31,A -85,B 0,C 180,E1 12066.732,E2 12066.732} C_VEL
LIN {X 0,Y 516.649,Z 707.31,A -85,B 0,C 180,E1 12071.845,E2 12071.845} C_VEL
LIN {X 0,Y 516.296,Z 707.31,A -85,B 0,C 180,E1 12077.065,E2 12077.065} C_VEL
LIN {X 0,Y 516.111,Z 707.31,A -85,B 0,C 180,E1 12082.436,E2 12082.436} C_VEL
LIN {X 0,Y 516.063,Z 707.31,A -85,B 0,C 180,E1 12088.243,E2 12088.243} C_VEL
LIN {X 0,Y 515.945,Z 707.31,A -85,B 0,C 180,E1 12093.917,E2 12093.917} C_VEL
LIN {X 0,Y 515.848,Z 707.31,A -85,B 0,C 180,E1 12100.258,E2 12100.258} C_VEL
LIN {X 0,Y 515.858,Z 707.31,A -85,B 0,C 180,E1 12103.587,E2 12103.587} C_VEL
LIN {X 0,Y 518.481,Z 713.184,A -85,B 0,C 180,E1 12103.999,E2 12103.999} C_VEL
LIN {X 0,Y 544.387,Z 759.077,A -85,B 0,C 180,E1 12107.482,E2 12107.482} C_VEL
LIN {X 0,Y 558.408,Z 790.581,A -85,B 0,C 180,E1 12109.521,E2 12109.521} C_VEL
LIN {X 0,Y 554.039,Z 834.69,A -85,B 0,C 180,E1 12110.873,E2 12110.873} C_VEL
LIN {X 0,Y 547.844,Z 880.425,A -85,B 0,C 180,E1 12113.012,E2 12113.012} C_VEL
LIN {X 0,Y 540.765,Z 924.05,A -85,B 0,C 180,E1 12115.911,E2 12115.911} C_VEL
LIN {X 0,Y 533.66,Z 963.891,A -85,B 0,C 180,E1 12119.513,E2 12119.513} C_VEL
LIN {X 0,Y 527.284,Z 999.167,A -85,B 0,C 180,E1 12123.776,E2 12123.776} C_VEL
LIN {X 0,Y 523.031,Z 1024.776,A -85,B 0,C 180,E1 12127.834,E2 12127.834} C_VEL
LIN {X 0,Y 517.815,Z 1033.729,A -85,B 0,C 180,E1 12129.393,E2 12129.393} C_VEL
LIN {X 0,Y 512.851,Z 1041.955,A -85,B 0,C 180,E1 12131.024,E2 12131.024} C_VEL
LIN {X 0,Y 510.739,Z 1060.038,A -85,B 0,C 180,E1 12135.83,E2 12135.83} C_VEL
LIN {X 0,Y 509.802,Z 1072.501,A -85,B 0,C 180,E1 12140.59,E2 12140.59} C_VEL
LIN {X 0,Y 509.525,Z 1079.202,A -85,B 0,C 180,E1 12144.88,E2 12144.88} C_VEL
LIN {X 0,Y 509.516,Z 1082.11,A -85,B 0,C 180,E1 12149.999,E2 12149.999} C_VEL
LIN {X 0,Y 509.524,Z 1079.198,A -85,B 0,C 180,E1 12155.118,E2 12155.118} C_VEL
LIN {X 0,Y 509.68,Z 1072.496,A -85,B 0,C 180,E1 12159.411,E2 12159.411} C_VEL
LIN {X 0,Y 510.834,Z 1058.716,A -85,B 0,C 180,E1 12164.604,E2 12164.604} C_VEL
LIN {X 0,Y 513.186,Z 1040.361,A -85,B 0,C 180,E1 12169.356,E2 12169.356} C_VEL
LIN {X 0,Y 517.201,Z 1014.985,A -85,B 0,C 180,E1 12174.217,E2 12174.217} C_VEL
LIN {X 0,Y 522.886,Z 984.866,A -85,B 0,C 180,E1 12178.567,E2 12178.567} C_VEL
LIN {X 0,Y 529.619,Z 949.905,A -85,B 0,C 180,E1 12182.428,E2 12182.428} C_VEL
LIN {X 0,Y 537.295,Z 909.474,A -85,B 0,C 180,E1 12185.772,E2 12185.772} C_VEL
LIN {X 0,Y 544.72,Z 864.502,A -85,B 0,C 180,E1 12188.476,E2 12188.476} C_VEL
LIN {X 0,Y 550.678,Z 819.999,A -85,B 0,C 180,E1 12190.319,E2 12190.319} C_VEL
LIN {X 0,Y 552.744,Z 790.846,A -85,B 0,C 180,E1 12191.231,E2 12191.231} C_VEL
LIN {X 0,Y 535.192,Z 754.045,A -85,B 0,C 180,E1 12193.929,E2 12193.929} C_VEL
LIN {X 0,Y 510.375,Z 713.052,A -85,B 0,C 180,E1 12197.598,E2 12197.598} C_VEL
LIN {X 0,Y 507.869,Z 707.31,A -85,B 0,C 180,E1 12198.103,E2 12198.103} C_VEL
LIN {X 0,Y 507.986,Z 707.31,A -85,B 0,C 180,E1 12203.652,E2 12203.652} C_VEL
LIN {X 0,Y 508.162,Z 707.31,A -85,B 0,C 180,E1 12209.86,E2 12209.86} C_VEL
LIN {X 0,Y 508.13,Z 707.31,A -85,B 0,C 180,E1 12215.325,E2 12215.325} C_VEL
LIN {X 0,Y 508.27,Z 707.31,A -85,B 0,C 180,E1 12220.858,E2 12220.858} C_VEL
LIN {X 0,Y 508.562,Z 707.31,A -85,B 0,C 180,E1 12226.212,E2 12226.212} C_VEL
LIN {X 0,Y 508.933,Z 707.31,A -85,B 0,C 180,E1 12231.441,E2 12231.441} C_VEL
LIN {X 0,Y 509.085,Z 707.31,A -85,B 0,C 180,E1 12238.297,E2 12238.297} C_VEL
LIN {X 0,Y 508.852,Z 707.31,A -85,B 0,C 180,E1 12245.129,E2 12245.129} C_VEL
LIN {X 0,Y 508.658,Z 707.31,A -85,B 0,C 180,E1 12252.04,E2 12252.04} C_VEL
LIN {X 0,Y 508.354,Z 707.31,A -85,B 0,C 180,E1 12257.465,E2 12257.465} C_VEL
LIN {X 0,Y 508.281,Z 707.31,A -85,B 0,C 180,E1 12262.807,E2 12262.807} C_VEL
LIN {X 0,Y 508.005,Z 707.31,A -85,B 0,C 180,E1 12268.511,E2 12268.511} C_VEL
LIN {X 0,Y 507.893,Z 707.31,A -85,B 0,C 180,E1 12274.538,E2 12274.538} C_VEL
LIN {X 0,Y 507.984,Z 707.694,A -85,B 0,C 180,E1 12280.32,E2 12280.32} C_VEL
LIN {X 0,Y 510.801,Z 713.342,A -85,B 0,C 180,E1 12280.795,E2 12280.795} C_VEL
LIN {X 0,Y 534.255,Z 753.158,A -85,B 0,C 180,E1 12284.397,E2 12284.397} C_VEL
LIN {X 0,Y 550.093,Z 788.327,A -85,B 0,C 180,E1 12287.19,E2 12287.19} C_VEL
LIN {X 0,Y 551.587,Z 795.088,A -85,B 0,C 180,E1 12287.601,E2 12287.601} C_VEL
LIN {X 0,Y 545.702,Z 840.884,A -85,B 0,C 180,E1 12289.506,E2 12289.506} C_VEL
LIN {X 0,Y 538.813,Z 882.985,A -85,B 0,C 180,E1 12292.032,E2 12292.032} C_VEL
LIN {X 0,Y 531.734,Z 920.483,A -85,B 0,C 180,E1 12295.075,E2 12295.075} C_VEL
LIN {X 0,Y 524.856,Z 954.414,A -85,B 0,C 180,E1 12298.688,E2 12298.688} C_VEL
LIN {X 0,Y 518.778,Z 985.016,A -85,B 0,C 180,E1 12302.966,E2 12302.966} C_VEL
LIN {X 0,Y 514.119,Z 1011.225,A -85,B 0,C 180,E1 12307.857,E2 12307.857} C_VEL
LIN {X 0,Y 511.36,Z 1030.457,A -85,B 0,C 180,E1 12312.763,E2 12312.763} C_VEL
LIN {X 0,Y 509.968,Z 1044.473,A -85,B 0,C 180,E1 12317.995,E2 12317.995} C_VEL
LIN {X 0,Y 509.457,Z 1051.599,A -85,B 0,C 180,E1 12322.308,E2 12322.308} C_VEL
LIN {X 0,Y 509.293,Z 1054.655,A -85,B 0,C 180,E1 12326.589,E2 12326.589} C_VEL
LIN {X 0,Y 509.572,Z 1054.452,A -85,B 0,C 180,E1 12330.001,E2 12330.001} C_VEL
LIN {X 0,Y 509.635,Z 1049.491,A -85,B 0,C 180,E1 12335.119,E2 12335.119} C_VEL
LIN {X 0,Y 510.388,Z 1038.857,A -85,B 0,C 180,E1 12340.263,E2 12340.263} C_VEL
LIN {X 0,Y 512.15,Z 1023.745,A -85,B 0,C 180,E1 12345.006,E2 12345.006} C_VEL
LIN {X 0,Y 515.507,Z 1002.32,A -85,B 0,C 180,E1 12349.827,E2 12349.827} C_VEL
LIN {X 0,Y 520.953,Z 972.707,A -85,B 0,C 180,E1 12354.719,E2 12354.719} C_VEL
LIN {X 0,Y 527.77,Z 938.08,A -85,B 0,C 180,E1 12358.968,E2 12358.968} C_VEL
LIN {X 0,Y 535.207,Z 898.987,A -85,B 0,C 180,E1 12362.546,E2 12362.546} C_VEL
LIN {X 0,Y 542.424,Z 856.117,A -85,B 0,C 180,E1 12365.431,E2 12365.431} C_VEL
LIN {X 0,Y 548.59,Z 810.945,A -85,B 0,C 180,E1 12367.576,E2 12367.576} C_VEL
LIN {X 0,Y 550.132,Z 791.758,A -85,B 0,C 180,E1 12368.295,E2 12368.295} C_VEL
LIN {X 0,Y 532.438,Z 751.361,A -85,B 0,C 180,E1 12371.314,E2 12371.314} C_VEL
LIN {X 0,Y 509.996,Z 712.626,A -85,B 0,C 180,E1 12374.554,E2 12374.554} C_VEL
LIN {X 0,Y 507.936,Z 707.31,A -85,B 0,C 180,E1 12374.944,E2 12374.944} C_VEL
LIN {X 0,Y 507.917,Z 707.31,A -85,B 0,C 180,E1 12381.201,E2 12381.201} C_VEL
LIN {X 0,Y 508.036,Z 707.31,A -85,B 0,C 180,E1 12387.523,E2 12387.523} C_VEL
LIN {X 0,Y 508.134,Z 707.31,A -85,B 0,C 180,E1 12393.47,E2 12393.47} C_VEL
LIN {X 0,Y 508.215,Z 707.31,A -85,B 0,C 180,E1 12399.031,E2 12399.031} C_VEL
LIN {X 0,Y 508.538,Z 707.31,A -85,B 0,C 180,E1 12404.44,E2 12404.44} C_VEL
LIN {X 0,Y 508.876,Z 707.31,A -85,B 0,C 180,E1 12409.704,E2 12409.704} C_VEL
LIN {X 0,Y 509.055,Z 707.31,A -85,B 0,C 180,E1 12414.873,E2 12414.873} C_VEL
LIN {X 0,Y 509.084,Z 707.31,A -85,B 0,C 180,E1 12421.703,E2 12421.703} C_VEL
LIN {X 0,Y 508.946,Z 707.31,A -85,B 0,C 180,E1 12428.559,E2 12428.559} C_VEL
LIN {X 0,Y 508.574,Z 707.31,A -85,B 0,C 180,E1 12433.787,E2 12433.787} C_VEL
LIN {X 0,Y 508.279,Z 707.31,A -85,B 0,C 180,E1 12439.141,E2 12439.141} C_VEL
LIN {X 0,Y 508.141,Z 707.31,A -85,B 0,C 180,E1 12444.674,E2 12444.674} C_VEL
LIN {X 0,Y 508.138,Z 707.31,A -85,B 0,C 180,E1 12450.459,E2 12450.459} C_VEL
LIN {X 0,Y 507.983,Z 707.31,A -85,B 0,C 180,E1 12456.625,E2 12456.625} C_VEL
LIN {X 0,Y 507.919,Z 707.31,A -85,B 0,C 180,E1 12462.655,E2 12462.655} C_VEL
LIN {X 0,Y 510.564,Z 713.21,A -85,B 0,C 180,E1 12463.106,E2 12463.106} C_VEL
LIN {X 0,Y 536.342,Z 758.088,A -85,B 0,C 180,E1 12466.697,E2 12466.697} C_VEL
LIN {X 0,Y 552.082,Z 792.169,A -85,B 0,C 180,E1 12469.033,E2 12469.033} C_VEL
LIN {X 0,Y 547.647,Z 835.599,A -85,B 0,C 180,E1 12470.4,E2 12470.4} C_VEL
LIN {X 0,Y 541.29,Z 880.828,A -85,B 0,C 180,E1 12472.544,E2 12472.544} C_VEL
LIN {X 0,Y 533.787,Z 925.016,A -85,B 0,C 180,E1 12475.528,E2 12475.528} C_VEL
LIN {X 0,Y 526.461,Z 964.458,A -85,B 0,C 180,E1 12479.159,E2 12479.159} C_VEL
LIN {X 0,Y 519.895,Z 999.165,A -85,B 0,C 180,E1 12483.419,E2 12483.419} C_VEL
LIN {X 0,Y 514.873,Z 1028.336,A -85,B 0,C 180,E1 12488.191,E2 12488.191} C_VEL
LIN {X 0,Y 512.851,Z 1041.955,A -85,B 0,C 180,E1 12491.024,E2 12491.024} C_VEL
LIN {X 0,Y 507.977,Z 1049.441,A -85,B 0,C 180,E1 12492.717,E2 12492.717} C_VEL
LIN {X 0,Y 503.297,Z 1056.184,A -85,B 0,C 180,E1 12494.479,E2 12494.479} C_VEL
LIN {X 0,Y 502.057,Z 1070.331,A -85,B 0,C 180,E1 12499.565,E2 12499.565} C_VEL
LIN {X 0,Y 501.601,Z 1077.985,A -85,B 0,C 180,E1 12503.929,E2 12503.929} C_VEL
LIN {X 0,Y 501.503,Z 1081.554,A -85,B 0,C 180,E1 12508.268,E2 12508.268} C_VEL
LIN {X 0,Y 501.673,Z 1081.558,A -85,B 0,C 180,E1 12511.73,E2 12511.73} C_VEL
LIN {X 0,Y 501.629,Z 1076.762,A -85,B 0,C 180,E1 12516.94,E2 12516.94} C_VEL
LIN {X 0,Y 502.208,Z 1067.824,A -85,B 0,C 180,E1 12521.56,E2 12521.56} C_VEL
LIN {X 0,Y 503.97,Z 1050.928,A -85,B 0,C 180,E1 12527.047,E2 12527.047} C_VEL
LIN {X 0,Y 507.551,Z 1026.964,A -85,B 0,C 180,E1 12532.435,E2 12532.435} C_VEL
LIN {X 0,Y 512.939,Z 997.863,A -85,B 0,C 180,E1 12537.244,E2 12537.244} C_VEL
LIN {X 0,Y 520.305,Z 962.406,A -85,B 0,C 180,E1 12541.617,E2 12541.617} C_VEL
LIN {X 0,Y 528.221,Z 922.969,A -85,B 0,C 180,E1 12545.256,E2 12545.256} C_VEL
LIN {X 0,Y 535.966,Z 880.536,A -85,B 0,C 180,E1 12548.136,E2 12548.136} C_VEL
LIN {X 0,Y 542.659,Z 835.893,A -85,B 0,C 180,E1 12550.284,E2 12550.284} C_VEL
LIN {X 0,Y 546.626,Z 793.704,A -85,B 0,C 180,E1 12551.708,E2 12551.708} C_VEL
LIN {X 0,Y 528.925,Z 756.262,A -85,B 0,C 180,E1 12554.551,E2 12554.551} C_VEL
LIN {X 0,Y 505.577,Z 718.093,A -85,B 0,C 180,E1 12558.105,E2 12558.105} C_VEL
LIN {X 0,Y 500.002,Z 708.24,A -85,B 0,C 180,E1 12559.054,E2 12559.054} C_VEL
LIN {X 0,Y 499.933,Z 707.31,A -85,B 0,C 180,E1 12559.269,E2 12559.269} C_VEL
LIN {X 0,Y 500.079,Z 707.31,A -85,B 0,C 180,E1 12564.902,E2 12564.902} C_VEL
LIN {X 0,Y 500.24,Z 707.31,A -85,B 0,C 180,E1 12571.461,E2 12571.461} C_VEL
LIN {X 0,Y 500.216,Z 707.31,A -85,B 0,C 180,E1 12576.811,E2 12576.811} C_VEL
LIN {X 0,Y 500.428,Z 707.31,A -85,B 0,C 180,E1 12582.376,E2 12582.376} C_VEL
LIN {X 0,Y 500.769,Z 707.31,A -85,B 0,C 180,E1 12587.774,E2 12587.774} C_VEL
LIN {X 0,Y 501.037,Z 707.31,A -85,B 0,C 180,E1 12593.055,E2 12593.055} C_VEL
LIN {X 0,Y 501.074,Z 707.31,A -85,B 0,C 180,E1 12600.003,E2 12600.003} C_VEL
LIN {X 0,Y 500.944,Z 707.31,A -85,B 0,C 180,E1 12605.21,E2 12605.21} C_VEL
LIN {X 0,Y 500.722,Z 707.31,A -85,B 0,C 180,E1 12612.234,E2 12612.234} C_VEL
LIN {X 0,Y 500.452,Z 707.31,A -85,B 0,C 180,E1 12617.629,E2 12617.629} C_VEL
LIN {X 0,Y 500.315,Z 707.31,A -85,B 0,C 180,E1 12623.191,E2 12623.191} C_VEL
LIN {X 0,Y 500.078,Z 707.31,A -85,B 0,C 180,E1 12629.006,E2 12629.006} C_VEL
LIN {X 0,Y 499.965,Z 707.31,A -85,B 0,C 180,E1 12635.165,E2 12635.165} C_VEL
LIN {X 0,Y 500.037,Z 707.862,A -85,B 0,C 180,E1 12639.275,E2 12639.275} C_VEL
LIN {X 0,Y 502.913,Z 713.419,A -85,B 0,C 180,E1 12639.78,E2 12639.78} C_VEL
LIN {X 0,Y 526.563,Z 752.78,A -85,B 0,C 180,E1 12643.552,E2 12643.552} C_VEL
LIN {X 0,Y 542.971,Z 788.733,A -85,B 0,C 180,E1 12646.526,E2 12646.526} C_VEL
LIN {X 0,Y 545.375,Z 797.57,A -85,B 0,C 180,E1 12647.131,E2 12647.131} C_VEL
LIN {X 0,Y 539.342,Z 842.698,A -85,B 0,C 180,E1 12649.051,E2 12649.051} C_VEL
LIN {X 0,Y 531.958,Z 885.658,A -85,B 0,C 180,E1 12651.685,E2 12651.685} C_VEL
LIN {X 0,Y 524.093,Z 925.482,A -85,B 0,C 180,E1 12655.04,E2 12655.04} C_VEL
LIN {X 0,Y 516.77,Z 959.712,A -85,B 0,C 180,E1 12658.88,E2 12658.88} C_VEL
LIN {X 0,Y 510.657,Z 988.828,A -85,B 0,C 180,E1 12663.175,E2 12663.175} C_VEL
LIN {X 0,Y 506.385,Z 1012.313,A -85,B 0,C 180,E1 12667.734,E2 12667.734} C_VEL
LIN {X 0,Y 503.418,Z 1032.014,A -85,B 0,C 180,E1 12672.933,E2 12672.933} C_VEL
LIN {X 0,Y 502.112,Z 1044.631,A -85,B 0,C 180,E1 12677.804,E2 12677.804} C_VEL
LIN {X 0,Y 501.574,Z 1051.782,A -85,B 0,C 180,E1 12682.187,E2 12682.187} C_VEL
LIN {X 0,Y 501.393,Z 1054.861,A -85,B 0,C 180,E1 12686.535,E2 12686.535} C_VEL
LIN {X 0,Y 501.672,Z 1054.679,A -85,B 0,C 180,E1 12690.001,E2 12690.001} C_VEL
LIN {X 0,Y 501.762,Z 1049.738,A -85,B 0,C 180,E1 12695.199,E2 12695.199} C_VEL
LIN {X 0,Y 502.583,Z 1039.133,A -85,B 0,C 180,E1 12700.424,E2 12700.424} C_VEL
LIN {X 0,Y 504.436,Z 1024.052,A -85,B 0,C 180,E1 12705.241,E2 12705.241} C_VEL
LIN {X 0,Y 508.182,Z 1001.596,A -85,B 0,C 180,E1 12710.335,E2 12710.335} C_VEL
LIN {X 0,Y 513.693,Z 973.079,A -85,B 0,C 180,E1 12715.092,E2 12715.092} C_VEL
LIN {X 0,Y 520.522,Z 939.808,A -85,B 0,C 180,E1 12719.255,E2 12719.255} C_VEL
LIN {X 0,Y 528.182,Z 901.274,A -85,B 0,C 180,E1 12722.867,E2 12722.867} C_VEL
LIN {X 0,Y 535.738,Z 858.479,A -85,B 0,C 180,E1 12725.816,E2 12725.816} C_VEL
LIN {X 0,Y 542.161,Z 813.428,A -85,B 0,C 180,E1 12728.008,E2 12728.008} C_VEL
LIN {X 0,Y 543.676,Z 794.111,A -85,B 0,C 180,E1 12728.774,E2 12728.774} C_VEL
LIN {X 0,Y 526.136,Z 753.828,A -85,B 0,C 180,E1 12731.882,E2 12731.882} C_VEL
LIN {X 0,Y 502.521,Z 713.093,A -85,B 0,C 180,E1 12735.431,E2 12735.431} C_VEL
LIN {X 0,Y 500.005,Z 707.31,A -85,B 0,C 180,E1 12735.92,E2 12735.92} C_VEL
LIN {X 0,Y 499.979,Z 707.31,A -85,B 0,C 180,E1 12742.004,E2 12742.004} C_VEL
LIN {X 0,Y 500.096,Z 707.31,A -85,B 0,C 180,E1 12748.046,E2 12748.046} C_VEL
LIN {X 0,Y 500.179,Z 707.31,A -85,B 0,C 180,E1 12752.967,E2 12752.967} C_VEL
LIN {X 0,Y 500.299,Z 707.31,A -85,B 0,C 180,E1 12758.683,E2 12758.683} C_VEL
LIN {X 0,Y 500.61,Z 707.31,A -85,B 0,C 180,E1 12764.187,E2 12764.187} C_VEL
LIN {X 0,Y 500.968,Z 707.31,A -85,B 0,C 180,E1 12769.54,E2 12769.54} C_VEL
LIN {X 0,Y 501.17,Z 707.31,A -85,B 0,C 180,E1 12774.792,E2 12774.792} C_VEL
LIN {X 0,Y 501.171,Z 707.31,A -85,B 0,C 180,E1 12781.73,E2 12781.73} C_VEL
LIN {X 0,Y 501.05,Z 707.31,A -85,B 0,C 180,E1 12788.694,E2 12788.694} C_VEL
LIN {X 0,Y 500.612,Z 707.31,A -85,B 0,C 180,E1 12794.377,E2 12794.377} C_VEL
LIN {X 0,Y 500.266,Z 707.31,A -85,B 0,C 180,E1 12800.106,E2 12800.106} C_VEL
LIN {X 0,Y 500.206,Z 707.31,A -85,B 0,C 180,E1 12805.092,E2 12805.092} C_VEL
LIN {X 0,Y 500.152,Z 707.31,A -85,B 0,C 180,E1 12810.999,E2 12810.999} C_VEL
LIN {X 0,Y 499.976,Z 707.31,A -85,B 0,C 180,E1 12817.31,E2 12817.31} C_VEL
LIN {X 0,Y 500.004,Z 708.122,A -85,B 0,C 180,E1 12821.741,E2 12821.741} C_VEL
LIN {X 0,Y 529.545,Z 759.551,A -85,B 0,C 180,E1 12826.057,E2 12826.057} C_VEL
LIN {X 0,Y 545.797,Z 795.442,A -85,B 0,C 180,E1 12828.589,E2 12828.589} C_VEL
LIN {X 0,Y 541.074,Z 838.179,A -85,B 0,C 180,E1 12829.986,E2 12829.986} C_VEL
LIN {X 0,Y 534.707,Z 881.496,A -85,B 0,C 180,E1 12832.082,E2 12832.082} C_VEL
LIN {X 0,Y 527.107,Z 924.657,A -85,B 0,C 180,E1 12835.028,E2 12835.028} C_VEL
LIN {X 0,Y 519.491,Z 963.801,A -85,B 0,C 180,E1 12838.657,E2 12838.657} C_VEL
LIN {X 0,Y 512.667,Z 998.396,A -85,B 0,C 180,E1 12842.938,E2 12842.938} C_VEL
LIN {X 0,Y 507.306,Z 1027.891,A -85,B 0,C 180,E1 12847.812,E2 12847.812} C_VEL
LIN {X 0,Y 503.946,Z 1050.781,A -85,B 0,C 180,E1 12852.95,E2 12852.95} C_VEL
LIN {X 0,Y 503.297,Z 1056.184,A -85,B 0,C 180,E1 12854.479,E2 12854.479} C_VEL
LIN {X 0,Y 498.771,Z 1062.141,A -85,B 0,C 180,E1 12856.294,E2 12856.294} C_VEL
LIN {X 0,Y 494.383,Z 1067.318,A -85,B 0,C 180,E1 12858.168,E2 12858.168} C_VEL
LIN {X 0,Y 493.764,Z 1076.531,A -85,B 0,C 180,E1 12862.948,E2 12862.948} C_VEL
LIN {X 0,Y 493.631,Z 1081.343,A -85,B 0,C 180,E1 12868.24,E2 12868.24} C_VEL
LIN {X 0,Y 493.792,Z 1081.348,A -85,B 0,C 180,E1 12871.758,E2 12871.758} C_VEL
LIN {X 0,Y 493.733,Z 1076.559,A -85,B 0,C 180,E1 12877.051,E2 12877.051} C_VEL
LIN {X 0,Y 494.338,Z 1067.783,A -85,B 0,C 180,E1 12881.684,E2 12881.684} C_VEL
LIN {X 0,Y 496.211,Z 1050.746,A -85,B 0,C 180,E1 12887.322,E2 12887.322} C_VEL
LIN {X 0,Y 500.045,Z 1026.804,A -85,B 0,C 180,E1 12892.791,E2 12892.791} C_VEL
LIN {X 0,Y 505.79,Z 997.311,A -85,B 0,C 180,E1 12897.727,E2 12897.727} C_VEL
LIN {X 0,Y 513.409,Z 962.307,A -85,B 0,C 180,E1 12902.092,E2 12902.092} C_VEL
LIN {X 0,Y 521.674,Z 922.827,A -85,B 0,C 180,E1 12905.774,E2 12905.774} C_VEL
LIN {X 0,Y 529.665,Z 880.625,A -85,B 0,C 180,E1 12908.666,E2 12908.666} C_VEL
LIN {X 0,Y 536.613,Z 835.969,A -85,B 0,C 180,E1 12910.833,E2 12910.833} C_VEL
LIN {X 0,Y 540.637,Z 796.702,A -85,B 0,C 180,E1 12912.182,E2 12912.182} C_VEL
LIN {X 0,Y 523.377,Z 760.053,A -85,B 0,C 180,E1 12915.079,E2 12915.079} C_VEL
LIN {X 0,Y 499.142,Z 719.776,A -85,B 0,C 180,E1 12918.92,E2 12918.92} C_VEL
LIN {X 0,Y 492.091,Z 708.382,A -85,B 0,C 180,E1 12920.153,E2 12920.153} C_VEL
LIN {X 0,Y 492.028,Z 707.31,A -85,B 0,C 180,E1 12920.35,E2 12920.35} C_VEL
LIN {X 0,Y 492.144,Z 707.31,A -85,B 0,C 180,E1 12926.345,E2 12926.345} C_VEL
LIN {X 0,Y 492.277,Z 707.31,A -85,B 0,C 180,E1 12932.504,E2 12932.504} C_VEL
LIN {X 0,Y 492.307,Z 707.31,A -85,B 0,C 180,E1 12938.326,E2 12938.326} C_VEL
LIN {X 0,Y 492.589,Z 707.31,A -85,B 0,C 180,E1 12943.93,E2 12943.93} C_VEL
LIN {X 0,Y 493.022,Z 707.31,A -85,B 0,C 180,E1 12949.598,E2 12949.598} C_VEL
LIN {X 0,Y 492.984,Z 707.31,A -85,B 0,C 180,E1 12954.712,E2 12954.712} C_VEL
LIN {X 0,Y 493.185,Z 707.31,A -85,B 0,C 180,E1 12960.003,E2 12960.003} C_VEL
LIN {X 0,Y 493.023,Z 707.31,A -85,B 0,C 180,E1 12965.294,E2 12965.294} C_VEL
LIN {X 0,Y 492.784,Z 707.31,A -85,B 0,C 180,E1 12972.434,E2 12972.434} C_VEL
LIN {X 0,Y 492.51,Z 707.31,A -85,B 0,C 180,E1 12977.923,E2 12977.923} C_VEL
LIN {X 0,Y 492.397,Z 707.31,A -85,B 0,C 180,E1 12983.587,E2 12983.587} C_VEL
LIN {X 0,Y 492.098,Z 707.31,A -85,B 0,C 180,E1 12989.522,E2 12989.522} C_VEL
LIN {X 0,Y 491.988,Z 707.31,A -85,B 0,C 180,E1 12995.823,E2 12995.823} C_VEL
LIN {X 0,Y 492.061,Z 707.349,A -85,B 0,C 180,E1 12998.153,E2 12998.153} C_VEL
LIN {X 0,Y 494.543,Z 713.034,A -85,B 0,C 180,E1 12998.633,E2 12998.633} C_VEL
LIN {X 0,Y 516.164,Z 747.448,A -85,B 0,C 180,E1 13002.201,E2 13002.201} C_VEL
LIN {X 0,Y 534.128,Z 784.639,A -85,B 0,C 180,E1 13005.469,E2 13005.469} C_VEL
LIN {X 0,Y 539.166,Z 800.384,A -85,B 0,C 180,E1 13006.668,E2 13006.668} C_VEL
LIN {X 0,Y 533.203,Z 842.99,A -85,B 0,C 180,E1 13008.506,E2 13008.506} C_VEL
LIN {X 0,Y 525.491,Z 886.355,A -85,B 0,C 180,E1 13011.192,E2 13011.192} C_VEL
LIN {X 0,Y 517.398,Z 925.732,A -85,B 0,C 180,E1 13014.548,E2 13014.548} C_VEL
LIN {X 0,Y 509.41,Z 961.511,A -85,B 0,C 180,E1 13018.629,E2 13018.629} C_VEL
LIN {X 0,Y 502.686,Z 992.428,A -85,B 0,C 180,E1 13023.358,E2 13023.358} C_VEL
LIN {X 0,Y 497.882,Z 1017.559,A -85,B 0,C 180,E1 13028.578,E2 13028.578} C_VEL
LIN {X 0,Y 495.316,Z 1034.806,A -85,B 0,C 180,E1 13033.562,E2 13033.562} C_VEL
LIN {X 0,Y 494.155,Z 1046.385,A -85,B 0,C 180,E1 13038.398,E2 13038.398} C_VEL
LIN {X 0,Y 493.637,Z 1052.82,A -85,B 0,C 180,E1 13042.947,E2 13042.947} C_VEL
LIN {X 0,Y 493.53,Z 1055.287,A -85,B 0,C 180,E1 13048.241,E2 13048.241} C_VEL
LIN {X 0,Y 493.691,Z 1053.894,A -85,B 0,C 180,E1 13051.76,E2 13051.76} C_VEL
LIN {X 0,Y 494.029,Z 1047.103,A -85,B 0,C 180,E1 13057.049,E2 13057.049} C_VEL
LIN {X 0,Y 495.17,Z 1035.974,A -85,B 0,C 180,E1 13061.883,E2 13061.883} C_VEL
LIN {X 0,Y 497.743,Z 1018.186,A -85,B 0,C 180,E1 13067.09,E2 13067.09} C_VEL
LIN {X 0,Y 502.445,Z 992.673,A -85,B 0,C 180,E1 13072.383,E2 13072.383} C_VEL
LIN {X 0,Y 508.804,Z 962.382,A -85,B 0,C 180,E1 13077.014,E2 13077.014} C_VEL
LIN {X 0,Y 516.549,Z 926.262,A -85,B 0,C 180,E1 13081.136,E2 13081.136} C_VEL
LIN {X 0,Y 524.455,Z 886.742,A -85,B 0,C 180,E1 13084.494,E2 13084.494} C_VEL
LIN {X 0,Y 531.767,Z 843.576,A -85,B 0,C 180,E1 13087.177,E2 13087.177} C_VEL
LIN {X 0,Y 537.624,Z 797.733,A -85,B 0,C 180,E1 13089.167,E2 13089.167} C_VEL
LIN {X 0,Y 521.087,Z 758.815,A -85,B 0,C 180,E1 13092.262,E2 13092.262} C_VEL
LIN {X 0,Y 498.711,Z 719.388,A -85,B 0,C 180,E1 13095.768,E2 13095.768} C_VEL
LIN {X 0,Y 492.183,Z 708.353,A -85,B 0,C 180,E1 13096.829,E2 13096.829} C_VEL
LIN {X 0,Y 492.093,Z 707.31,A -85,B 0,C 180,E1 13096.964,E2 13096.964} C_VEL
LIN {X 0,Y 492.045,Z 707.31,A -85,B 0,C 180,E1 13103.203,E2 13103.203} C_VEL
LIN {X 0,Y 492.184,Z 707.31,A -85,B 0,C 180,E1 13109.555,E2 13109.555} C_VEL
LIN {X 0,Y 492.261,Z 707.31,A -85,B 0,C 180,E1 13114.467,E2 13114.467} C_VEL
LIN {X 0,Y 492.429,Z 707.31,A -85,B 0,C 180,E1 13120.211,E2 13120.211} C_VEL
LIN {X 0,Y 492.836,Z 707.31,A -85,B 0,C 180,E1 13125.757,E2 13125.757} C_VEL
LIN {X 0,Y 493.067,Z 707.31,A -85,B 0,C 180,E1 13131.86,E2 13131.86} C_VEL
LIN {X 0,Y 493.069,Z 707.31,A -85,B 0,C 180,E1 13136.473,E2 13136.473} C_VEL
LIN {X 0,Y 493.259,Z 707.31,A -85,B 0,C 180,E1 13141.757,E2 13141.757} C_VEL
LIN {X 0,Y 493.123,Z 707.31,A -85,B 0,C 180,E1 13148.835,E2 13148.835} C_VEL
LIN {X 0,Y 492.721,Z 707.31,A -85,B 0,C 180,E1 13154.24,E2 13154.24} C_VEL
LIN {X 0,Y 492.394,Z 707.31,A -85,B 0,C 180,E1 13159.784,E2 13159.784} C_VEL
LIN {X 0,Y 492.253,Z 707.31,A -85,B 0,C 180,E1 13165.526,E2 13165.526} C_VEL
LIN {X 0,Y 492.212,Z 707.31,A -85,B 0,C 180,E1 13171.556,E2 13171.556} C_VEL
LIN {X 0,Y 492.069,Z 707.31,A -85,B 0,C 180,E1 13178.015,E2 13178.015} C_VEL
LIN {X 0,Y 492.043,Z 707.363,A -85,B 0,C 180,E1 13180.714,E2 13180.714} C_VEL
LIN {X 0,Y 494.377,Z 712.863,A -85,B 0,C 180,E1 13181.132,E2 13181.132} C_VEL
LIN {X 0,Y 518.444,Z 752.884,A -85,B 0,C 180,E1 13184.757,E2 13184.757} C_VEL
LIN {X 0,Y 537.578,Z 793.022,A -85,B 0,C 180,E1 13187.761,E2 13187.761} C_VEL
LIN {X 0,Y 539.402,Z 799.69,A -85,B 0,C 180,E1 13188.154,E2 13188.154} C_VEL
LIN {X 0,Y 534.143,Z 843.657,A -85,B 0,C 180,E1 13189.684,E2 13189.684} C_VEL
LIN {X 0,Y 527.458,Z 886.244,A -85,B 0,C 180,E1 13191.859,E2 13191.859} C_VEL
LIN {X 0,Y 520.069,Z 926.136,A -85,B 0,C 180,E1 13194.668,E2 13194.668} C_VEL
LIN {X 0,Y 512.255,Z 964.678,A -85,B 0,C 180,E1 13198.317,E2 13198.317} C_VEL
LIN {X 0,Y 505.266,Z 998.591,A -85,B 0,C 180,E1 13202.589,E2 13202.589} C_VEL
LIN {X 0,Y 500.043,Z 1026.266,A -85,B 0,C 180,E1 13207.202,E2 13207.202} C_VEL
LIN {X 0,Y 496.401,Z 1048.762,A -85,B 0,C 180,E1 13212.224,E2 13212.224} C_VEL
LIN {X 0,Y 494.589,Z 1064.694,A -85,B 0,C 180,E1 13217.165,E2 13217.165} C_VEL
LIN {X 0,Y 494.383,Z 1067.318,A -85,B 0,C 180,E1 13218.168,E2 13218.168} C_VEL
LIN {X 0,Y 490.198,Z 1071.788,A -85,B 0,C 180,E1 13220.076,E2 13220.076} C_VEL
LIN {X 0,Y 485.968,Z 1075.177,A -85,B 0,C 180,E1 13222.046,E2 13222.046} C_VEL
LIN {X 0,Y 485.741,Z 1080.267,A -85,B 0,C 180,E1 13226.617,E2 13226.617} C_VEL
LIN {X 0,Y 485.888,Z 1081.139,A -85,B 0,C 180,E1 13231.786,E2 13231.786} C_VEL
LIN {X 0,Y 485.839,Z 1076.359,A -85,B 0,C 180,E1 13237.166,E2 13237.166} C_VEL
LIN {X 0,Y 486.496,Z 1067.351,A -85,B 0,C 180,E1 13241.974,E2 13241.974} C_VEL
LIN {X 0,Y 488.463,Z 1050.567,A -85,B 0,C 180,E1 13247.606,E2 13247.606} C_VEL
LIN {X 0,Y 492.283,Z 1027.817,A -85,B 0,C 180,E1 13252.921,E2 13252.921} C_VEL
LIN {X 0,Y 498.168,Z 998.979,A -85,B 0,C 180,E1 13257.891,E2 13257.891} C_VEL
LIN {X 0,Y 505.602,Z 966.112,A -85,B 0,C 180,E1 13262.14,E2 13262.14} C_VEL
LIN {X 0,Y 513.633,Z 929.781,A -85,B 0,C 180,E1 13265.706,E2 13265.706} C_VEL
LIN {X 0,Y 521.533,Z 890.436,A -85,B 0,C 180,E1 13268.614,E2 13268.614} C_VEL
LIN {X 0,Y 528.893,Z 847.19,A -85,B 0,C 180,E1 13270.934,E2 13270.934} C_VEL
LIN {X 0,Y 534.738,Z 800.148,A -85,B 0,C 180,E1 13272.645,E2 13272.645} C_VEL
LIN {X 0,Y 518.106,Z 764.061,A -85,B 0,C 180,E1 13275.586,E2 13275.586} C_VEL
LIN {X 0,Y 495.313,Z 725.876,A -85,B 0,C 180,E1 13279.308,E2 13279.308} C_VEL
LIN {X 0,Y 484.361,Z 709.293,A -85,B 0,C 180,E1 13281.269,E2 13281.269} C_VEL
LIN {X 0,Y 484.123,Z 707.31,A -85,B 0,C 180,E1 13281.493,E2 13281.493} C_VEL
LIN {X 0,Y 484.226,Z 707.31,A -85,B 0,C 180,E1 13287.862,E2 13287.862} C_VEL
LIN {X 0,Y 484.323,Z 707.31,A -85,B 0,C 180,E1 13294.025,E2 13294.025} C_VEL
LIN {X 0,Y 484.452,Z 707.31,A -85,B 0,C 180,E1 13299.878,E2 13299.878} C_VEL
LIN {X 0,Y 484.817,Z 707.31,A -85,B 0,C 180,E1 13305.686,E2 13305.686} C_VEL
LIN {X 0,Y 485.186,Z 707.31,A -85,B 0,C 180,E1 13311.019,E2 13311.019} C_VEL
LIN {X 0,Y 485.355,Z 707.31,A -85,B 0,C 180,E1 13318.214,E2 13318.214} C_VEL
LIN {X 0,Y 485.123,Z 707.31,A -85,B 0,C 180,E1 13325.38,E2 13325.38} C_VEL
LIN {X 0,Y 484.847,Z 707.31,A -85,B 0,C 180,E1 13332.641,E2 13332.641} C_VEL
LIN {X 0,Y 484.57,Z 707.31,A -85,B 0,C 180,E1 13338.227,E2 13338.227} C_VEL
LIN {X 0,Y 484.416,Z 707.31,A -85,B 0,C 180,E1 13344,E2 13344} C_VEL
LIN {X 0,Y 484.179,Z 707.31,A -85,B 0,C 180,E1 13350.055,E2 13350.055} C_VEL
LIN {X 0,Y 484.126,Z 707.81,A -85,B 0,C 180,E1 13356.994,E2 13356.994} C_VEL
LIN {X 0,Y 486.967,Z 713.383,A -85,B 0,C 180,E1 13357.55,E2 13357.55} C_VEL
LIN {X 0,Y 509.024,Z 748.223,A -85,B 0,C 180,E1 13361.356,E2 13361.356} C_VEL
LIN {X 0,Y 527.172,Z 785.406,A -85,B 0,C 180,E1 13364.774,E2 13364.774} C_VEL
LIN {X 0,Y 533.067,Z 802.438,A -85,B 0,C 180,E1 13366.164,E2 13366.164} C_VEL
LIN {X 0,Y 526.882,Z 844.797,A -85,B 0,C 180,E1 13368.034,E2 13368.034} C_VEL
LIN {X 0,Y 519.12,Z 886.671,A -85,B 0,C 180,E1 13370.658,E2 13370.658} C_VEL
LIN {X 0,Y 510.541,Z 926.845,A -85,B 0,C 180,E1 13374.124,E2 13374.124} C_VEL
LIN {X 0,Y 502.293,Z 962.128,A -85,B 0,C 180,E1 13378.215,E2 13378.215} C_VEL
LIN {X 0,Y 495.334,Z 992.516,A -85,B 0,C 180,E1 13382.931,E2 13382.931} C_VEL
LIN {X 0,Y 490.549,Z 1016.459,A -85,B 0,C 180,E1 13387.942,E2 13387.942} C_VEL
LIN {X 0,Y 487.751,Z 1033.63,A -85,B 0,C 180,E1 13392.834,E2 13392.834} C_VEL
LIN {X 0,Y 486.421,Z 1044.956,A -85,B 0,C 180,E1 13397.405,E2 13397.405} C_VEL
LIN {X 0,Y 485.821,Z 1052.149,A -85,B 0,C 180,E1 13401.932,E2 13401.932} C_VEL
LIN {X 0,Y 485.578,Z 1055.397,A -85,B 0,C 180,E1 13407.084,E2 13407.084} C_VEL
LIN {X 0,Y 485.794,Z 1054.119,A -85,B 0,C 180,E1 13411.788,E2 13411.788} C_VEL
LIN {X 0,Y 486.164,Z 1047.356,A -85,B 0,C 180,E1 13417.163,E2 13417.163} C_VEL
LIN {X 0,Y 487.39,Z 1035.934,A -85,B 0,C 180,E1 13422.187,E2 13422.187} C_VEL
LIN {X 0,Y 490.153,Z 1017.755,A -85,B 0,C 180,E1 13427.544,E2 13427.544} C_VEL
LIN {X 0,Y 494.983,Z 993.018,A -85,B 0,C 180,E1 13432.739,E2 13432.739} C_VEL
LIN {X 0,Y 501.662,Z 962.762,A -85,B 0,C 180,E1 13437.431,E2 13437.431} C_VEL
LIN {X 0,Y 509.668,Z 926.692,A -85,B 0,C 180,E1 13441.605,E2 13441.605} C_VEL
LIN {X 0,Y 517.933,Z 887.275,A -85,B 0,C 180,E1 13444.987,E2 13444.987} C_VEL
LIN {X 0,Y 525.503,Z 844.114,A -85,B 0,C 180,E1 13447.698,E2 13447.698} C_VEL
LIN {X 0,Y 531.269,Z 800.507,A -85,B 0,C 180,E1 13449.629,E2 13449.629} C_VEL
LIN {X 0,Y 515.661,Z 763.043,A -85,B 0,C 180,E1 13452.715,E2 13452.715} C_VEL
LIN {X 0,Y 494.488,Z 725.175,A -85,B 0,C 180,E1 13456.176,E2 13456.176} C_VEL
LIN {X 0,Y 484.311,Z 708.803,A -85,B 0,C 180,E1 13457.869,E2 13457.869} C_VEL
LIN {X 0,Y 484.156,Z 707.31,A -85,B 0,C 180,E1 13458.038,E2 13458.038} C_VEL
LIN {X 0,Y 484.127,Z 707.31,A -85,B 0,C 180,E1 13464.475,E2 13464.475} C_VEL
LIN {X 0,Y 484.282,Z 707.31,A -85,B 0,C 180,E1 13471.185,E2 13471.185} C_VEL
LIN {X 0,Y 484.441,Z 707.31,A -85,B 0,C 180,E1 13477.949,E2 13477.949} C_VEL
LIN {X 0,Y 484.731,Z 707.31,A -85,B 0,C 180,E1 13483.655,E2 13483.655} C_VEL
LIN {X 0,Y 485.115,Z 707.31,A -85,B 0,C 180,E1 13489.194,E2 13489.194} C_VEL
LIN {X 0,Y 485.361,Z 707.31,A -85,B 0,C 180,E1 13494.622,E2 13494.622} C_VEL
LIN {X 0,Y 485.369,Z 707.31,A -85,B 0,C 180,E1 13501.786,E2 13501.786} C_VEL
LIN {X 0,Y 485.199,Z 707.31,A -85,B 0,C 180,E1 13508.981,E2 13508.981} C_VEL
LIN {X 0,Y 484.799,Z 707.31,A -85,B 0,C 180,E1 13514.478,E2 13514.478} C_VEL
LIN {X 0,Y 484.44,Z 707.31,A -85,B 0,C 180,E1 13520.206,E2 13520.206} C_VEL
LIN {X 0,Y 484.333,Z 707.31,A -85,B 0,C 180,E1 13525.975,E2 13525.975} C_VEL
LIN {X 0,Y 484.227,Z 707.31,A -85,B 0,C 180,E1 13532.33,E2 13532.33} C_VEL
LIN {X 0,Y 484.121,Z 707.31,A -85,B 0,C 180,E1 13538.754,E2 13538.754} C_VEL
LIN {X 0,Y 484.137,Z 707.337,A -85,B 0,C 180,E1 13539.656,E2 13539.656} C_VEL
LIN {X 0,Y 486.614,Z 713.072,A -85,B 0,C 180,E1 13540.12,E2 13540.12} C_VEL
LIN {X 0,Y 510.514,Z 752.183,A -85,B 0,C 180,E1 13543.871,E2 13543.871} C_VEL
LIN {X 0,Y 529.665,Z 791.674,A -85,B 0,C 180,E1 13546.965,E2 13546.965} C_VEL
LIN {X 0,Y 533.172,Z 802.303,A -85,B 0,C 180,E1 13547.673,E2 13547.673} C_VEL
LIN {X 0,Y 527.579,Z 846.683,A -85,B 0,C 180,E1 13549.271,E2 13549.271} C_VEL
LIN {X 0,Y 520.559,Z 889.181,A -85,B 0,C 180,E1 13551.52,E2 13551.52} C_VEL
LIN {X 0,Y 513.032,Z 927.745,A -85,B 0,C 180,E1 13554.31,E2 13554.31} C_VEL
LIN {X 0,Y 505.296,Z 964.409,A -85,B 0,C 180,E1 13557.836,E2 13557.836} C_VEL
LIN {X 0,Y 498.056,Z 998.113,A -85,B 0,C 180,E1 13562.128,E2 13562.128} C_VEL
LIN {X 0,Y 492.272,Z 1027.269,A -85,B 0,C 180,E1 13567.08,E2 13567.08} C_VEL
LIN {X 0,Y 488.452,Z 1050.271,A -85,B 0,C 180,E1 13572.392,E2 13572.392} C_VEL
LIN {X 0,Y 486.512,Z 1067.192,A -85,B 0,C 180,E1 13578.017,E2 13578.017} C_VEL
LIN {X 0,Y 485.968,Z 1075.177,A -85,B 0,C 180,E1 13582.046,E2 13582.046} C_VEL
LIN {X 0,Y 481.794,Z 1077.903,A -85,B 0,C 180,E1 13584.041,E2 13584.041} C_VEL
LIN {X 0,Y 477.835,Z 1079.685,A -85,B 0,C 180,E1 13586.078,E2 13586.078} C_VEL
LIN {X 0,Y 477.951,Z 1081.266,A -85,B 0,C 180,E1 13589.999,E2 13589.999} C_VEL
LIN {X 0,Y 477.931,Z 1078.379,A -85,B 0,C 180,E1 13595.458,E2 13595.458} C_VEL
LIN {X 0,Y 478.189,Z 1071.753,A -85,B 0,C 180,E1 13600.008,E2 13600.008} C_VEL
LIN {X 0,Y 479.568,Z 1058.994,A -85,B 0,C 180,E1 13605.226,E2 13605.226} C_VEL
LIN {X 0,Y 482.248,Z 1041.452,A -85,B 0,C 180,E1 13610.221,E2 13610.221} C_VEL
LIN {X 0,Y 487.179,Z 1016.227,A -85,B 0,C 180,E1 13615.476,E2 13615.476} C_VEL
LIN {X 0,Y 494.325,Z 984.888,A -85,B 0,C 180,E1 13620.312,E2 13620.312} C_VEL
LIN {X 0,Y 502.777,Z 948.628,A -85,B 0,C 180,E1 13624.5,E2 13624.5} C_VEL
LIN {X 0,Y 511.617,Z 908.756,A -85,B 0,C 180,E1 13627.923,E2 13627.923} C_VEL
LIN {X 0,Y 520.244,Z 863.56,A -85,B 0,C 180,E1 13630.723,E2 13630.723} C_VEL
LIN {X 0,Y 527.396,Z 816.709,A -85,B 0,C 180,E1 13632.687,E2 13632.687} C_VEL
LIN {X 0,Y 528.34,Z 802.01,A -85,B 0,C 180,E1 13633.223,E2 13633.223} C_VEL
LIN {X 0,Y 511.111,Z 764.738,A -85,B 0,C 180,E1 13636.395,E2 13636.395} C_VEL
LIN {X 0,Y 487.764,Z 726.16,A -85,B 0,C 180,E1 13640.372,E2 13640.372} C_VEL
LIN {X 0,Y 478.43,Z 712.84,A -85,B 0,C 180,E1 13642.101,E2 13642.101} C_VEL
LIN {X 0,Y 476.157,Z 707.31,A -85,B 0,C 180,E1 13642.714,E2 13642.714} C_VEL
LIN {X 0,Y 476.327,Z 707.31,A -85,B 0,C 180,E1 13649.405,E2 13649.405} C_VEL
LIN {X 0,Y 476.433,Z 707.31,A -85,B 0,C 180,E1 13655.579,E2 13655.579} C_VEL
LIN {X 0,Y 476.647,Z 707.31,A -85,B 0,C 180,E1 13662.51,E2 13662.51} C_VEL
LIN {X 0,Y 477.138,Z 707.31,A -85,B 0,C 180,E1 13669.018,E2 13669.018} C_VEL
LIN {X 0,Y 477.2,Z 707.31,A -85,B 0,C 180,E1 13674.537,E2 13674.537} C_VEL
LIN {X 0,Y 477.395,Z 707.31,A -85,B 0,C 180,E1 13680.003,E2 13680.003} C_VEL
LIN {X 0,Y 477.2,Z 707.31,A -85,B 0,C 180,E1 13685.47,E2 13685.47} C_VEL
LIN {X 0,Y 476.942,Z 707.31,A -85,B 0,C 180,E1 13692.854,E2 13692.854} C_VEL
LIN {X 0,Y 476.65,Z 707.31,A -85,B 0,C 180,E1 13698.541,E2 13698.541} C_VEL
LIN {X 0,Y 476.478,Z 707.31,A -85,B 0,C 180,E1 13704.425,E2 13704.425} C_VEL
LIN {X 0,Y 476.185,Z 707.31,A -85,B 0,C 180,E1 13710.77,E2 13710.77} C_VEL
LIN {X 0,Y 476.152,Z 707.31,A -85,B 0,C 180,E1 13715.729,E2 13715.729} C_VEL
LIN {X 0,Y 478.486,Z 712.905,A -85,B 0,C 180,E1 13716.243,E2 13716.243} C_VEL
LIN {X 0,Y 498.724,Z 743.584,A -85,B 0,C 180,E1 13719.919,E2 13719.919} C_VEL
LIN {X 0,Y 517.517,Z 779.945,A -85,B 0,C 180,E1 13723.473,E2 13723.473} C_VEL
LIN {X 0,Y 526.912,Z 805.223,A -85,B 0,C 180,E1 13725.675,E2 13725.675} C_VEL
LIN {X 0,Y 520.591,Z 846.581,A -85,B 0,C 180,E1 13727.549,E2 13727.549} C_VEL
LIN {X 0,Y 512.724,Z 887.439,A -85,B 0,C 180,E1 13730.144,E2 13730.144} C_VEL
LIN {X 0,Y 503.747,Z 927.752,A -85,B 0,C 180,E1 13733.67,E2 13733.67} C_VEL
LIN {X 0,Y 494.883,Z 964.202,A -85,B 0,C 180,E1 13737.991,E2 13737.991} C_VEL
LIN {X 0,Y 487.772,Z 993.922,A -85,B 0,C 180,E1 13742.727,E2 13742.727} C_VEL
LIN {X 0,Y 482.764,Z 1017.798,A -85,B 0,C 180,E1 13747.873,E2 13747.873} C_VEL
LIN {X 0,Y 479.811,Z 1035.101,A -85,B 0,C 180,E1 13753.014,E2 13753.014} C_VEL
LIN {X 0,Y 478.433,Z 1046.912,A -85,B 0,C 180,E1 13758.12,E2 13758.12} C_VEL
LIN {X 0,Y 477.861,Z 1053.198,A -85,B 0,C 180,E1 13762.713,E2 13762.713} C_VEL
LIN {X 0,Y 477.739,Z 1055.718,A -85,B 0,C 180,E1 13768.183,E2 13768.183} C_VEL
LIN {X 0,Y 477.9,Z 1054.343,A -85,B 0,C 180,E1 13771.818,E2 13771.818} C_VEL
LIN {X 0,Y 478.289,Z 1047.608,A -85,B 0,C 180,E1 13777.282,E2 13777.282} C_VEL
LIN {X 0,Y 479.605,Z 1036.227,A -85,B 0,C 180,E1 13782.383,E2 13782.383} C_VEL
LIN {X 0,Y 482.495,Z 1018.063,A -85,B 0,C 180,E1 13787.833,E2 13787.833} C_VEL
LIN {X 0,Y 487.522,Z 993.58,A -85,B 0,C 180,E1 13793.066,E2 13793.066} C_VEL
LIN {X 0,Y 494.571,Z 963.137,A -85,B 0,C 180,E1 13797.858,E2 13797.858} C_VEL
LIN {X 0,Y 502.897,Z 927.196,A -85,B 0,C 180,E1 13802.072,E2 13802.072} C_VEL
LIN {X 0,Y 511.433,Z 887.746,A -85,B 0,C 180,E1 13805.498,E2 13805.498} C_VEL
LIN {X 0,Y 519.527,Z 843.271,A -85,B 0,C 180,E1 13808.305,E2 13808.305} C_VEL
LIN {X 0,Y 524.899,Z 803.232,A -85,B 0,C 180,E1 13810.109,E2 13810.109} C_VEL
LIN {X 0,Y 509.766,Z 766.348,A -85,B 0,C 180,E1 13813.249,E2 13813.249} C_VEL
LIN {X 0,Y 490.171,Z 730.712,A -85,B 0,C 180,E1 13816.611,E2 13816.611} C_VEL
LIN {X 0,Y 476.345,Z 708.771,A -85,B 0,C 180,E1 13818.993,E2 13818.993} C_VEL
LIN {X 0,Y 476.152,Z 707.31,A -85,B 0,C 180,E1 13819.2,E2 13819.2} C_VEL
LIN {X 0,Y 476.255,Z 707.31,A -85,B 0,C 180,E1 13825.823,E2 13825.823} C_VEL
LIN {X 0,Y 476.391,Z 707.31,A -85,B 0,C 180,E1 13831.497,E2 13831.497} C_VEL
LIN {X 0,Y 476.485,Z 707.31,A -85,B 0,C 180,E1 13837.561,E2 13837.561} C_VEL
LIN {X 0,Y 476.772,Z 707.31,A -85,B 0,C 180,E1 13843.374,E2 13843.374} C_VEL
LIN {X 0,Y 477.179,Z 707.31,A -85,B 0,C 180,E1 13849.897,E2 13849.897} C_VEL
LIN {X 0,Y 477.444,Z 707.31,A -85,B 0,C 180,E1 13854.533,E2 13854.533} C_VEL
LIN {X 0,Y 477.479,Z 707.31,A -85,B 0,C 180,E1 13861.815,E2 13861.815} C_VEL
LIN {X 0,Y 477.27,Z 707.31,A -85,B 0,C 180,E1 13869.131,E2 13869.131} C_VEL
LIN {X 0,Y 476.853,Z 707.31,A -85,B 0,C 180,E1 13874.725,E2 13874.725} C_VEL
LIN {X 0,Y 476.527,Z 707.31,A -85,B 0,C 180,E1 13880.472,E2 13880.472} C_VEL
LIN {X 0,Y 476.358,Z 707.31,A -85,B 0,C 180,E1 13887.032,E2 13887.032} C_VEL
LIN {X 0,Y 476.274,Z 707.31,A -85,B 0,C 180,E1 13892.741,E2 13892.741} C_VEL
LIN {X 0,Y 476.251,Z 707.703,A -85,B 0,C 180,E1 13898.551,E2 13898.551} C_VEL
LIN {X 0,Y 478.941,Z 713.263,A -85,B 0,C 180,E1 13899.064,E2 13899.064} C_VEL
LIN {X 0,Y 503.302,Z 752.759,A -85,B 0,C 180,E1 13903.056,E2 13903.056} C_VEL
LIN {X 0,Y 522.24,Z 791.605,A -85,B 0,C 180,E1 13906.229,E2 13906.229} C_VEL
LIN {X 0,Y 526.968,Z 804.226,A -85,B 0,C 180,E1 13907.164,E2 13907.164} C_VEL
LIN {X 0,Y 521.197,Z 848.553,A -85,B 0,C 180,E1 13908.799,E2 13908.799} C_VEL
LIN {X 0,Y 513.673,Z 892.195,A -85,B 0,C 180,E1 13911.177,E2 13911.177} C_VEL
LIN {X 0,Y 505.317,Z 932.681,A -85,B 0,C 180,E1 13914.229,E2 13914.229} C_VEL
LIN {X 0,Y 497.503,Z 967.973,A -85,B 0,C 180,E1 13917.787,E2 13917.787} C_VEL
LIN {X 0,Y 490.46,Z 999.413,A -85,B 0,C 180,E1 13921.929,E2 13921.929} C_VEL
LIN {X 0,Y 484.557,Z 1028.013,A -85,B 0,C 180,E1 13926.918,E2 13926.918} C_VEL
LIN {X 0,Y 480.736,Z 1050.012,A -85,B 0,C 180,E1 13932.1,E2 13932.1} C_VEL
LIN {X 0,Y 478.684,Z 1066.553,A -85,B 0,C 180,E1 13937.661,E2 13937.661} C_VEL
LIN {X 0,Y 477.982,Z 1076.082,A -85,B 0,C 180,E1 13942.713,E2 13942.713} C_VEL
LIN {X 0,Y 477.835,Z 1079.685,A -85,B 0,C 180,E1 13946.078,E2 13946.078} C_VEL
LIN {X 0,Y 474.009,Z 1080.909,A -85,B 0,C 180,E1 13948.126,E2 13948.126} C_VEL
LIN {X 0,Y 470.032,Z 1081.016,A -85,B 0,C 180,E1 13950.213,E2 13950.213} C_VEL
LIN {X 0,Y 470.043,Z 1078.177,A -85,B 0,C 180,E1 13955.549,E2 13955.549} C_VEL
LIN {X 0,Y 470.396,Z 1070.701,A -85,B 0,C 180,E1 13960.61,E2 13960.61} C_VEL
LIN {X 0,Y 472.182,Z 1056.048,A -85,B 0,C 180,E1 13966.428,E2 13966.428} C_VEL
LIN {X 0,Y 475.703,Z 1035.37,A -85,B 0,C 180,E1 13971.981,E2 13971.981} C_VEL
LIN {X 0,Y 481.732,Z 1007.553,A -85,B 0,C 180,E1 13977.39,E2 13977.39} C_VEL
LIN {X 0,Y 490.038,Z 973.618,A -85,B 0,C 180,E1 13982.237,E2 13982.237} C_VEL
LIN {X 0,Y 499.212,Z 935.574,A -85,B 0,C 180,E1 13986.272,E2 13986.272} C_VEL
LIN {X 0,Y 508.556,Z 893.251,A -85,B 0,C 180,E1 13989.561,E2 13989.561} C_VEL
LIN {X 0,Y 516.75,Z 848.836,A -85,B 0,C 180,E1 13992.025,E2 13992.025} C_VEL
LIN {X 0,Y 522.301,Z 805.035,A -85,B 0,C 180,E1 13993.724,E2 13993.724} C_VEL
LIN {X 0,Y 505.425,Z 767.967,A -85,B 0,C 180,E1 13997.003,E2 13997.003} C_VEL
LIN {X 0,Y 483.409,Z 731.518,A -85,B 0,C 180,E1 14000.89,E2 14000.89} C_VEL
LIN {X 0,Y 470.724,Z 713.083,A -85,B 0,C 180,E1 14003.35,E2 14003.35} C_VEL
LIN {X 0,Y 468.227,Z 707.31,A -85,B 0,C 180,E1 14004.008,E2 14004.008} C_VEL
LIN {X 0,Y 468.364,Z 707.31,A -85,B 0,C 180,E1 14008.827,E2 14008.827} C_VEL
LIN {X 0,Y 468.468,Z 707.31,A -85,B 0,C 180,E1 14015.136,E2 14015.136} C_VEL
LIN {X 0,Y 468.648,Z 707.31,A -85,B 0,C 180,E1 14021.138,E2 14021.138} C_VEL
LIN {X 0,Y 469.034,Z 707.31,A -85,B 0,C 180,E1 14026.932,E2 14026.932} C_VEL
LIN {X 0,Y 469.377,Z 707.31,A -85,B 0,C 180,E1 14032.584,E2 14032.584} C_VEL
LIN {X 0,Y 469.503,Z 707.31,A -85,B 0,C 180,E1 14040.003,E2 14040.003} C_VEL
LIN {X 0,Y 469.289,Z 707.31,A -85,B 0,C 180,E1 14045.563,E2 14045.563} C_VEL
LIN {X 0,Y 469.062,Z 707.31,A -85,B 0,C 180,E1 14051.18,E2 14051.18} C_VEL
LIN {X 0,Y 468.798,Z 707.31,A -85,B 0,C 180,E1 14056.917,E2 14056.917} C_VEL
LIN {X 0,Y 468.644,Z 707.31,A -85,B 0,C 180,E1 14062.835,E2 14062.835} C_VEL
LIN {X 0,Y 468.313,Z 707.31,A -85,B 0,C 180,E1 14069.112,E2 14069.112} C_VEL
LIN {X 0,Y 468.248,Z 707.361,A -85,B 0,C 180,E1 14074.415,E2 14074.415} C_VEL
LIN {X 0,Y 470.476,Z 712.797,A -85,B 0,C 180,E1 14074.935,E2 14074.935} C_VEL
LIN {X 0,Y 485.107,Z 734.081,A -85,B 0,C 180,E1 14077.76,E2 14077.76} C_VEL
LIN {X 0,Y 504.016,Z 766.944,A -85,B 0,C 180,E1 14081.35,E2 14081.35} C_VEL
LIN {X 0,Y 518.564,Z 800.466,A -85,B 0,C 180,E1 14084.539,E2 14084.539} C_VEL
LIN {X 0,Y 520.85,Z 807.801,A -85,B 0,C 180,E1 14085.169,E2 14085.169} C_VEL
LIN {X 0,Y 514.232,Z 848.848,A -85,B 0,C 180,E1 14087.078,E2 14087.078} C_VEL
LIN {X 0,Y 506.197,Z 888.892,A -85,B 0,C 180,E1 14089.673,E2 14089.673} C_VEL
LIN {X 0,Y 497.168,Z 927.886,A -85,B 0,C 180,E1 14093.125,E2 14093.125} C_VEL
LIN {X 0,Y 488.122,Z 963.674,A -85,B 0,C 180,E1 14097.397,E2 14097.397} C_VEL
LIN {X 0,Y 480.419,Z 994.373,A -85,B 0,C 180,E1 14102.345,E2 14102.345} C_VEL
LIN {X 0,Y 475.069,Z 1018.662,A -85,B 0,C 180,E1 14107.684,E2 14107.684} C_VEL
LIN {X 0,Y 471.883,Z 1036.574,A -85,B 0,C 180,E1 14113.201,E2 14113.201} C_VEL
LIN {X 0,Y 470.577,Z 1047.088,A -85,B 0,C 180,E1 14117.918,E2 14117.918} C_VEL
LIN {X 0,Y 469.971,Z 1053.389,A -85,B 0,C 180,E1 14122.59,E2 14122.59} C_VEL
LIN {X 0,Y 469.869,Z 1055.933,A -85,B 0,C 180,E1 14128.153,E2 14128.153} C_VEL
LIN {X 0,Y 470.003,Z 1054.567,A -85,B 0,C 180,E1 14131.849,E2 14131.849} C_VEL
LIN {X 0,Y 470.441,Z 1047.858,A -85,B 0,C 180,E1 14137.404,E2 14137.404} C_VEL
LIN {X 0,Y 471.708,Z 1037.289,A -85,B 0,C 180,E1 14142.313,E2 14142.313} C_VEL
LIN {X 0,Y 474.85,Z 1018.371,A -85,B 0,C 180,E1 14148.13,E2 14148.13} C_VEL
LIN {X 0,Y 480.195,Z 993.626,A -85,B 0,C 180,E1 14153.494,E2 14153.494} C_VEL
LIN {X 0,Y 487.492,Z 963.508,A -85,B 0,C 180,E1 14158.299,E2 14158.299} C_VEL
LIN {X 0,Y 496.278,Z 927.017,A -85,B 0,C 180,E1 14162.62,E2 14162.62} C_VEL
LIN {X 0,Y 505.269,Z 886.826,A -85,B 0,C 180,E1 14166.125,E2 14166.125} C_VEL
LIN {X 0,Y 513.377,Z 843.833,A -85,B 0,C 180,E1 14168.849,E2 14168.849} C_VEL
LIN {X 0,Y 518.72,Z 806.248,A -85,B 0,C 180,E1 14170.57,E2 14170.57} C_VEL
LIN {X 0,Y 503.88,Z 769.538,A -85,B 0,C 180,E1 14173.794,E2 14173.794} C_VEL
LIN {X 0,Y 485.409,Z 735.686,A -85,B 0,C 180,E1 14177.116,E2 14177.116} C_VEL
LIN {X 0,Y 470.031,Z 712.323,A -85,B 0,C 180,E1 14179.845,E2 14179.845} C_VEL
LIN {X 0,Y 468.222,Z 707.31,A -85,B 0,C 180,E1 14180.354,E2 14180.354} C_VEL
LIN {X 0,Y 468.355,Z 707.31,A -85,B 0,C 180,E1 14187.274,E2 14187.274} C_VEL
LIN {X 0,Y 468.459,Z 707.31,A -85,B 0,C 180,E1 14193.068,E2 14193.068} C_VEL
LIN {X 0,Y 468.665,Z 707.31,A -85,B 0,C 180,E1 14199.671,E2 14199.671} C_VEL
LIN {X 0,Y 469.066,Z 707.31,A -85,B 0,C 180,E1 14205.747,E2 14205.747} C_VEL
LIN {X 0,Y 469.336,Z 707.31,A -85,B 0,C 180,E1 14211.881,E2 14211.881} C_VEL
LIN {X 0,Y 469.402,Z 707.31,A -85,B 0,C 180,E1 14216.295,E2 14216.295} C_VEL
LIN {X 0,Y 469.58,Z 707.31,A -85,B 0,C 180,E1 14221.846,E2 14221.846} C_VEL
LIN {X 0,Y 469.391,Z 707.31,A -85,B 0,C 180,E1 14227.416,E2 14227.416} C_VEL
LIN {X 0,Y 469.048,Z 707.31,A -85,B 0,C 180,E1 14233.067,E2 14233.067} C_VEL
LIN {X 0,Y 468.656,Z 707.31,A -85,B 0,C 180,E1 14238.862,E2 14238.862} C_VEL
LIN {X 0,Y 468.458,Z 707.31,A -85,B 0,C 180,E1 14245.072,E2 14245.072} C_VEL
LIN {X 0,Y 468.367,Z 707.31,A -85,B 0,C 180,E1 14251.172,E2 14251.172} C_VEL
LIN {X 0,Y 468.288,Z 707.78,A -85,B 0,C 180,E1 14257.362,E2 14257.362} C_VEL
LIN {X 0,Y 471.051,Z 713.307,A -85,B 0,C 180,E1 14257.915,E2 14257.915} C_VEL
LIN {X 0,Y 494.915,Z 751.349,A -85,B 0,C 180,E1 14262.013,E2 14262.013} C_VEL
LIN {X 0,Y 513.879,Z 789.052,A -85,B 0,C 180,E1 14265.273,E2 14265.273} C_VEL
LIN {X 0,Y 520.683,Z 807.334,A -85,B 0,C 180,E1 14266.681,E2 14266.681} C_VEL
LIN {X 0,Y 514.758,Z 850.754,A -85,B 0,C 180,E1 14268.338,E2 14268.338} C_VEL
LIN {X 0,Y 507.081,Z 893.495,A -85,B 0,C 180,E1 14270.714,E2 14270.714} C_VEL
LIN {X 0,Y 498.105,Z 935.372,A -85,B 0,C 180,E1 14273.952,E2 14273.952} C_VEL
LIN {X 0,Y 489.316,Z 973.485,A -85,B 0,C 180,E1 14277.969,E2 14277.969} C_VEL
LIN {X 0,Y 481.667,Z 1006.282,A -85,B 0,C 180,E1 14282.604,E2 14282.604} C_VEL
LIN {X 0,Y 475.841,Z 1033.569,A -85,B 0,C 180,E1 14287.778,E2 14287.778} C_VEL
LIN {X 0,Y 472.269,Z 1054.469,A -85,B 0,C 180,E1 14293.214,E2 14293.214} C_VEL
LIN {X 0,Y 470.743,Z 1067.426,A -85,B 0,C 180,E1 14297.921,E2 14297.921} C_VEL
LIN {X 0,Y 470.055,Z 1077.09,A -85,B 0,C 180,E1 14303.52,E2 14303.52} C_VEL
LIN {X 0,Y 469.941,Z 1080.738,A -85,B 0,C 180,E1 14308.325,E2 14308.325} C_VEL
LIN {X 0,Y 470.032,Z 1081.016,A -85,B 0,C 180,E1 14310.213,E2 14310.213} C_VEL
LIN {X 0,Y 466.03,Z 1080.468,A -85,B 0,C 180,E1 14312.292,E2 14312.292} C_VEL
LIN {X 0,Y 462.068,Z 1079.017,A -85,B 0,C 180,E1 14314.401,E2 14314.401} C_VEL
LIN {X 0,Y 462.288,Z 1072.909,A -85,B 0,C 180,E1 14319.433,E2 14319.433} C_VEL
LIN {X 0,Y 463.505,Z 1061.68,A -85,B 0,C 180,E1 14324.677,E2 14324.677} C_VEL
LIN {X 0,Y 466.693,Z 1042.8,A -85,B 0,C 180,E1 14330.497,E2 14330.497} C_VEL
LIN {X 0,Y 472.411,Z 1016.344,A -85,B 0,C 180,E1 14336.255,E2 14336.255} C_VEL
LIN {X 0,Y 480.187,Z 984.999,A -85,B 0,C 180,E1 14341.252,E2 14341.252} C_VEL
LIN {X 0,Y 489.583,Z 948.103,A -85,B 0,C 180,E1 14345.611,E2 14345.611} C_VEL
LIN {X 0,Y 499.214,Z 907.638,A -85,B 0,C 180,E1 14349.137,E2 14349.137} C_VEL
LIN {X 0,Y 508.208,Z 864.041,A -85,B 0,C 180,E1 14351.875,E2 14351.875} C_VEL
LIN {X 0,Y 515.887,Z 816.85,A -85,B 0,C 180,E1 14353.887,E2 14353.887} C_VEL
LIN {X 0,Y 516.304,Z 808.041,A -85,B 0,C 180,E1 14354.238,E2 14354.238} C_VEL
LIN {X 0,Y 500.084,Z 772.008,A -85,B 0,C 180,E1 14357.544,E2 14357.544} C_VEL
LIN {X 0,Y 479.365,Z 737.106,A -85,B 0,C 180,E1 14361.37,E2 14361.37} C_VEL
LIN {X 0,Y 462.981,Z 713.234,A -85,B 0,C 180,E1 14364.691,E2 14364.691} C_VEL
LIN {X 0,Y 460.332,Z 708.049,A -85,B 0,C 180,E1 14365.314,E2 14365.314} C_VEL
LIN {X 0,Y 460.466,Z 707.31,A -85,B 0,C 180,E1 14370.423,E2 14370.423} C_VEL
LIN {X 0,Y 460.661,Z 707.31,A -85,B 0,C 180,E1 14377.084,E2 14377.084} C_VEL
LIN {X 0,Y 460.823,Z 707.31,A -85,B 0,C 180,E1 14382.789,E2 14382.789} C_VEL
LIN {X 0,Y 461.256,Z 707.31,A -85,B 0,C 180,E1 14388.635,E2 14388.635} C_VEL
LIN {X 0,Y 461.415,Z 707.31,A -85,B 0,C 180,E1 14394.349,E2 14394.349} C_VEL
LIN {X 0,Y 461.599,Z 707.31,A -85,B 0,C 180,E1 14400.003,E2 14400.003} C_VEL
LIN {X 0,Y 461.365,Z 707.31,A -85,B 0,C 180,E1 14405.658,E2 14405.658} C_VEL
LIN {X 0,Y 461.145,Z 707.31,A -85,B 0,C 180,E1 14411.375,E2 14411.375} C_VEL
LIN {X 0,Y 460.814,Z 707.31,A -85,B 0,C 180,E1 14417.512,E2 14417.512} C_VEL
LIN {X 0,Y 460.683,Z 707.31,A -85,B 0,C 180,E1 14423.253,E2 14423.253} C_VEL
LIN {X 0,Y 460.362,Z 707.31,A -85,B 0,C 180,E1 14429.592,E2 14429.592} C_VEL
LIN {X 0,Y 460.391,Z 708.162,A -85,B 0,C 180,E1 14433.033,E2 14433.033} C_VEL
LIN {X 0,Y 463.418,Z 713.558,A -85,B 0,C 180,E1 14433.729,E2 14433.729} C_VEL
LIN {X 0,Y 484.796,Z 745.682,A -85,B 0,C 180,E1 14438.033,E2 14438.033} C_VEL
LIN {X 0,Y 502.701,Z 779.424,A -85,B 0,C 180,E1 14441.692,E2 14441.692} C_VEL
LIN {X 0,Y 514.762,Z 809.92,A -85,B 0,C 180,E1 14444.62,E2 14444.62} C_VEL
LIN {X 0,Y 507.749,Z 852.065,A -85,B 0,C 180,E1 14446.652,E2 14446.652} C_VEL
LIN {X 0,Y 499.434,Z 891.488,A -85,B 0,C 180,E1 14449.282,E2 14449.282} C_VEL
LIN {X 0,Y 490.111,Z 930.03,A -85,B 0,C 180,E1 14452.782,E2 14452.782} C_VEL
LIN {X 0,Y 481.106,Z 964.341,A -85,B 0,C 180,E1 14456.96,E2 14456.96} C_VEL
LIN {X 0,Y 473.206,Z 994.457,A -85,B 0,C 180,E1 14461.884,E2 14461.884} C_VEL
LIN {X 0,Y 467.399,Z 1019.376,A -85,B 0,C 180,E1 14467.455,E2 14467.455} C_VEL
LIN {X 0,Y 463.936,Z 1038.035,A -85,B 0,C 180,E1 14473.394,E2 14473.394} C_VEL
LIN {X 0,Y 462.568,Z 1048.803,A -85,B 0,C 180,E1 14478.665,E2 14478.665} C_VEL
LIN {X 0,Y 462.082,Z 1053.58,A -85,B 0,C 180,E1 14482.463,E2 14482.463} C_VEL
LIN {X 0,Y 461.967,Z 1056.148,A -85,B 0,C 180,E1 14488.121,E2 14488.121} C_VEL
LIN {X 0,Y 462.106,Z 1054.79,A -85,B 0,C 180,E1 14491.88,E2 14491.88} C_VEL
LIN {X 0,Y 462.566,Z 1048.107,A -85,B 0,C 180,E1 14497.531,E2 14497.531} C_VEL
LIN {X 0,Y 463.981,Z 1036.976,A -85,B 0,C 180,E1 14502.737,E2 14502.737} C_VEL
LIN {X 0,Y 467.223,Z 1018.678,A -85,B 0,C 180,E1 14508.436,E2 14508.436} C_VEL
LIN {X 0,Y 472.654,Z 994.68,A -85,B 0,C 180,E1 14513.748,E2 14513.748} C_VEL
LIN {X 0,Y 480.433,Z 963.876,A -85,B 0,C 180,E1 14518.753,E2 14518.753} C_VEL
LIN {X 0,Y 489.474,Z 927.883,A -85,B 0,C 180,E1 14523.079,E2 14523.079} C_VEL
LIN {X 0,Y 498.836,Z 887.492,A -85,B 0,C 180,E1 14526.649,E2 14526.649} C_VEL
LIN {X 0,Y 507.18,Z 844.763,A -85,B 0,C 180,E1 14529.388,E2 14529.388} C_VEL
LIN {X 0,Y 512.185,Z 808.435,A -85,B 0,C 180,E1 14531.125,E2 14531.125} C_VEL
LIN {X 0,Y 498.02,Z 772.847,A -85,B 0,C 180,E1 14534.349,E2 14534.349} C_VEL
LIN {X 0,Y 478.807,Z 737.125,A -85,B 0,C 180,E1 14537.978,E2 14537.978} C_VEL
LIN {X 0,Y 462.231,Z 712.488,A -85,B 0,C 180,E1 14541.058,E2 14541.058} C_VEL
LIN {X 0,Y 460.286,Z 707.31,A -85,B 0,C 180,E1 14541.524,E2 14541.524} C_VEL
LIN {X 0,Y 460.433,Z 707.31,A -85,B 0,C 180,E1 14548.22,E2 14548.22} C_VEL
LIN {X 0,Y 460.547,Z 707.31,A -85,B 0,C 180,E1 14554.671,E2 14554.671} C_VEL
LIN {X 0,Y 460.758,Z 707.31,A -85,B 0,C 180,E1 14560.795,E2 14560.795} C_VEL
LIN {X 0,Y 461.217,Z 707.31,A -85,B 0,C 180,E1 14566.7,E2 14566.7} C_VEL
LIN {X 0,Y 461.5,Z 707.31,A -85,B 0,C 180,E1 14572.449,E2 14572.449} C_VEL
LIN {X 0,Y 461.331,Z 707.31,A -85,B 0,C 180,E1 14578.114,E2 14578.114} C_VEL
LIN {X 0,Y 461.377,Z 707.31,A -85,B 0,C 180,E1 14583.763,E2 14583.763} C_VEL
LIN {X 0,Y 461.376,Z 707.31,A -85,B 0,C 180,E1 14589.813,E2 14589.813} C_VEL
LIN {X 0,Y 460.983,Z 707.31,A -85,B 0,C 180,E1 14595.244,E2 14595.244} C_VEL
LIN {X 0,Y 460.633,Z 707.31,A -85,B 0,C 180,E1 14601.212,E2 14601.212} C_VEL
LIN {X 0,Y 460.517,Z 707.31,A -85,B 0,C 180,E1 14607.427,E2 14607.427} C_VEL
LIN {X 0,Y 460.338,Z 707.31,A -85,B 0,C 180,E1 14614.025,E2 14614.025} C_VEL
LIN {X 0,Y 460.365,Z 707.786,A -85,B 0,C 180,E1 14616.104,E2 14616.104} C_VEL
LIN {X 0,Y 462.986,Z 713.172,A -85,B 0,C 180,E1 14616.663,E2 14616.663} C_VEL
LIN {X 0,Y 485.493,Z 748.011,A -85,B 0,C 180,E1 14620.733,E2 14620.733} C_VEL
LIN {X 0,Y 505.033,Z 785.401,A -85,B 0,C 180,E1 14624.174,E2 14624.174} C_VEL
LIN {X 0,Y 514.445,Z 810.279,A -85,B 0,C 180,E1 14626.179,E2 14626.179} C_VEL
LIN {X 0,Y 508.448,Z 852.199,A -85,B 0,C 180,E1 14627.831,E2 14627.831} C_VEL
LIN {X 0,Y 500.498,Z 894.74,A -85,B 0,C 180,E1 14630.236,E2 14630.236} C_VEL
LIN {X 0,Y 491.284,Z 936.161,A -85,B 0,C 180,E1 14633.495,E2 14633.495} C_VEL
LIN {X 0,Y 482.38,Z 973.15,A -85,B 0,C 180,E1 14637.453,E2 14637.453} C_VEL
LIN {X 0,Y 474.376,Z 1005.977,A -85,B 0,C 180,E1 14642.147,E2 14642.147} C_VEL
LIN {X 0,Y 468.3,Z 1033.291,A -85,B 0,C 180,E1 14647.401,E2 14647.401} C_VEL
LIN {X 0,Y 464.504,Z 1054.211,A -85,B 0,C 180,E1 14652.925,E2 14652.925} C_VEL
LIN {X 0,Y 462.904,Z 1067.188,A -85,B 0,C 180,E1 14657.713,E2 14657.713} C_VEL
LIN {X 0,Y 462.171,Z 1076.863,A -85,B 0,C 180,E1 14663.409,E2 14663.409} C_VEL
LIN {X 0,Y 462.045,Z 1080.492,A -85,B 0,C 180,E1 14668.12,E2 14668.12} C_VEL
LIN {X 0,Y 462.205,Z 1080.512,A -85,B 0,C 180,E1 14671.878,E2 14671.878} C_VEL
LIN {X 0,Y 462.068,Z 1079.017,A -85,B 0,C 180,E1 14674.401,E2 14674.401} C_VEL
LIN {X 0,Y 458.192,Z 1077.089,A -85,B 0,C 180,E1 14676.515,E2 14676.515} C_VEL
LIN {X 0,Y 454.36,Z 1074.281,A -85,B 0,C 180,E1 14678.648,E2 14678.648} C_VEL
LIN {X 0,Y 455.543,Z 1062.694,A -85,B 0,C 180,E1 14684.447,E2 14684.447} C_VEL
LIN {X 0,Y 458.282,Z 1046.623,A -85,B 0,C 180,E1 14689.745,E2 14689.745} C_VEL
LIN {X 0,Y 463.177,Z 1023.94,A -85,B 0,C 180,E1 14695.17,E2 14695.17} C_VEL
LIN {X 0,Y 470.469,Z 995.427,A -85,B 0,C 180,E1 14700.22,E2 14700.22} C_VEL
LIN {X 0,Y 479.563,Z 961.097,A -85,B 0,C 180,E1 14704.763,E2 14704.763} C_VEL
LIN {X 0,Y 489.661,Z 921.812,A -85,B 0,C 180,E1 14708.601,E2 14708.601} C_VEL
LIN {X 0,Y 499.268,Z 879.585,A -85,B 0,C 180,E1 14711.601,E2 14711.601} C_VEL
LIN {X 0,Y 507.382,Z 835.691,A -85,B 0,C 180,E1 14713.795,E2 14713.795} C_VEL
LIN {X 0,Y 510.304,Z 811.104,A -85,B 0,C 180,E1 14714.767,E2 14714.767} C_VEL
LIN {X 0,Y 494.413,Z 775.066,A -85,B 0,C 180,E1 14718.179,E2 14718.179} C_VEL
LIN {X 0,Y 472.885,Z 738.649,A -85,B 0,C 180,E1 14722.352,E2 14722.352} C_VEL
LIN {X 0,Y 455.147,Z 713.285,A -85,B 0,C 180,E1 14726.148,E2 14726.148} C_VEL
LIN {X 0,Y 452.48,Z 708.484,A -85,B 0,C 180,E1 14726.809,E2 14726.809} C_VEL
LIN {X 0,Y 452.393,Z 707.31,A -85,B 0,C 180,E1 14726.868,E2 14726.868} C_VEL
LIN {X 0,Y 452.538,Z 707.31,A -85,B 0,C 180,E1 14732.047,E2 14732.047} C_VEL
LIN {X 0,Y 452.721,Z 707.31,A -85,B 0,C 180,E1 14738.399,E2 14738.399} C_VEL
LIN {X 0,Y 453.017,Z 707.31,A -85,B 0,C 180,E1 14744.482,E2 14744.482} C_VEL
LIN {X 0,Y 453.501,Z 707.31,A -85,B 0,C 180,E1 14750.386,E2 14750.386} C_VEL
LIN {X 0,Y 453.486,Z 707.31,A -85,B 0,C 180,E1 14756.171,E2 14756.171} C_VEL
LIN {X 0,Y 453.417,Z 707.31,A -85,B 0,C 180,E1 14761.919,E2 14761.919} C_VEL
LIN {X 0,Y 453.28,Z 707.31,A -85,B 0,C 180,E1 14767.688,E2 14767.688} C_VEL
LIN {X 0,Y 453.064,Z 707.31,A -85,B 0,C 180,E1 14774.077,E2 14774.077} C_VEL
LIN {X 0,Y 452.803,Z 707.31,A -85,B 0,C 180,E1 14780.436,E2 14780.436} C_VEL
LIN {X 0,Y 452.591,Z 707.31,A -85,B 0,C 180,E1 14785.806,E2 14785.806} C_VEL
LIN {X 0,Y 452.443,Z 707.314,A -85,B 0,C 180,E1 14791.483,E2 14791.483} C_VEL
LIN {X 0,Y 454.566,Z 712.676,A -85,B 0,C 180,E1 14792.056,E2 14792.056} C_VEL
LIN {X 0,Y 457.678,Z 716.726,A -85,B 0,C 180,E1 14792.764,E2 14792.764} C_VEL
LIN {X 0,Y 477.488,Z 746.114,A -85,B 0,C 180,E1 14796.948,E2 14796.948} C_VEL
LIN {X 0,Y 495.185,Z 778.929,A -85,B 0,C 180,E1 14800.713,E2 14800.713} C_VEL
LIN {X 0,Y 508.648,Z 812.857,A -85,B 0,C 180,E1 14804.093,E2 14804.093} C_VEL
LIN {X 0,Y 500.438,Z 859.65,A -85,B 0,C 180,E1 14806.467,E2 14806.467} C_VEL
LIN {X 0,Y 491.177,Z 900.74,A -85,B 0,C 180,E1 14809.424,E2 14809.424} C_VEL
LIN {X 0,Y 481.468,Z 938.462,A -85,B 0,C 180,E1 14813.132,E2 14813.132} C_VEL
LIN {X 0,Y 472.521,Z 970.755,A -85,B 0,C 180,E1 14817.371,E2 14817.371} C_VEL
LIN {X 0,Y 465.028,Z 997.972,A -85,B 0,C 180,E1 14822.097,E2 14822.097} C_VEL
LIN {X 0,Y 459.558,Z 1020.769,A -85,B 0,C 180,E1 14827.421,E2 14827.421} C_VEL
